KUKA KRL program: f1_Kuka_APT219T02S19.SRC

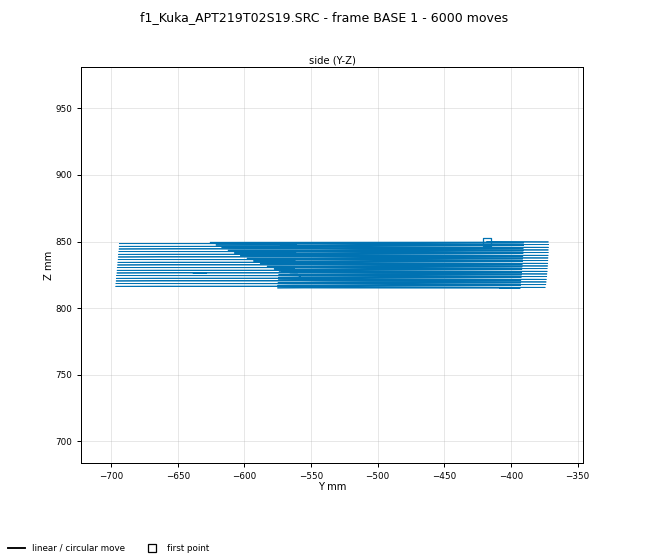
[picture p0: tool path of f1_Kuka_APT219T02S19.SRC in frame BASE 1, 6000 of 6001 moves have a stored position in this frame; points joined in program order, loops and branches not executed]
&ACCESS RVP
&REL 2
&PARAM TEMPLATE = C:\KRC\Roboter\Template\vorgabe
&PARAM EDITMASK = *
DEF f1_Kuka_APT219T02S19()


;FOLD INI;%{PE}%V3.2.0,%MKUKATPBASIS,%CINIT,%VCOMMON,%P
  ;FOLD BAS INI;%{E}%V3.2.0,%MKUKATPBASIS,%CINIT,%VINIT,%P
    GLOBAL INTERRUPT DECL 3 WHEN $STOPMESS==TRUE DO IR_STOPM ( )
    INTERRUPT ON 3
    BAS (#INITMOV,0 )
  ;ENDFOLD (BAS INI)
  ;FOLD USER INI;%{E}%V3.2.0,%MKUKATPUSER,%CINIT,%VINIT,%P
    ;Make your modifications here
  ;ENDFOLD (USER INI)
;ENDFOLD (INI)


;*** Make Null PTP Move
  PTP $pos_act

;*** Auto Load The Correct TOOL Data
  $tool=tool_data[2]

;*** Auto Load The Correct BASE Data
  $base=base_data[1]

  $ADVANCE = 5

;*** Restate Last Velocity
MMPM(30000.0)
SetRPM(8000)
LIN {X -0.097,Y -418.240,Z 849.890,A 0.000,B 0.000,C 90.000,E1 196.134} C_DIS
LIN {X -0.095,Y -415.487,Z 849.882,A 0.000,B 0.000,C 90.000,E1 194.773} C_DIS
LIN {X 0.056,Y -410.579,Z 849.869,A 0.000,B 0.000,C 90.000,E1 192.355} C_DIS
LIN {X -0.158,Y -407.973,Z 849.861,A 0.000,B 0.000,C 90.000,E1 191.007} C_DIS
LIN {X -0.079,Y -404.648,Z 849.851,A 0.000,B 0.000,C 90.000,E1 189.265} C_DIS
LIN {X -0.066,Y -401.875,Z 849.844,A 0.000,B 0.000,C 90.000,E1 187.871} C_DIS
LIN {X -0.071,Y -394.854,Z 849.822,A 0.000,B 0.000,C 90.000,E1 184.012} C_DIS
LIN {X 0.068,Y -390.052,Z 849.805,A 0.000,B 0.000,C 90.000,E1 180.802} C_DIS
LIN {X -0.073,Y -387.200,Z 849.793,A 0.000,B 0.000,C 90.000,E1 178.682} C_DIS
LIN {X 0.013,Y -383.709,Z 849.779,A 0.000,B 0.000,C 90.000,E1 176.159} C_DIS
LIN {X 0.052,Y -380.406,Z 849.765,A 0.000,B 0.000,C 90.000,E1 173.628} C_DIS
LIN {X -0.090,Y -378.246,Z 849.755,A 0.000,B 0.000,C 90.000,E1 171.837} C_DIS
LIN {X -0.103,Y -375.157,Z 849.738,A 0.000,B 0.000,C 90.000,E1 168.926} C_DIS
LIN {X -0.058,Y -372.815,Z 849.722,A 0.000,B 0.000,C 90.000,E1 165.992} C_DIS
LIN {X 0.084,Y -371.867,Z 849.706,A 0.000,B 0.000,C 90.000,E1 163.032} C_DIS
LIN {X 0.049,Y -371.826,Z 849.704,A 0.000,B 0.000,C 90.000,E1 162.670} C_DIS
LIN {X -0.054,Y -372.398,Z 849.698,A 0.000,B 0.000,C 90.000,E1 161.583} C_DIS
LIN {X -0.120,Y -372.933,Z 849.694,A 0.000,B 0.000,C 90.000,E1 160.859} C_DIS
LIN {X -0.003,Y -373.909,Z 849.690,A 0.000,B 0.000,C 90.000,E1 160.115} C_DIS
LIN {X -0.017,Y -374.079,Z 849.689,A 0.000,B 0.000,C 90.000,E1 159.934} C_DIS
LIN {X -0.070,Y -375.433,Z 849.685,A 0.000,B 0.000,C 90.000,E1 159.209} C_DIS
LIN {X 0.178,Y -376.512,Z 849.682,A 0.000,B 0.000,C 90.000,E1 158.773} C_DIS
LIN {X 0.157,Y -377.673,Z 849.680,A 0.000,B 0.000,C 90.000,E1 158.411} C_DIS
LIN {X -0.114,Y -379.654,Z 849.677,A 0.000,B 0.000,C 90.000,E1 157.922} C_DIS
LIN {X 0.023,Y -380.338,Z 849.676,A 0.000,B 0.000,C 90.000,E1 157.720} C_DIS
LIN {X -0.133,Y -381.711,Z 849.675,A 0.000,B 0.000,C 90.000,E1 157.486} C_DIS
LIN {X -0.008,Y -383.667,Z 849.673,A 0.000,B 0.000,C 90.000,E1 157.177} C_DIS
LIN {X -0.104,Y -387.727,Z 849.671,A 0.000,B 0.000,C 90.000,E1 156.719} C_DIS
LIN {X -0.011,Y -389.404,Z 849.670,A 0.000,B 0.000,C 90.000,E1 156.538} C_DIS
LIN {X -0.049,Y -392.267,Z 849.669,A 0.000,B 0.000,C 90.000,E1 156.357} C_DIS
LIN {X -0.038,Y -402.998,Z 849.666,A 0.000,B 0.000,C 90.000,E1 155.845} C_DIS
LIN {X 0.052,Y -407.988,Z 849.665,A 0.000,B 0.000,C 90.000,E1 155.665} C_DIS
LIN {X 0.056,Y -414.236,Z 849.663,A 0.000,B 0.000,C 90.000,E1 155.409} C_DIS
LIN {X -0.004,Y -424.366,Z 849.661,A 0.000,B 0.000,C 90.000,E1 154.973} C_DIS
LIN {X 0.156,Y -433.945,Z 849.658,A 0.000,B 0.000,C 90.000,E1 154.409} C_DIS
LIN {X -0.258,Y -437.088,Z 849.657,A 0.000,B 0.000,C 90.000,E1 154.280} C_DIS
LIN {X 0.137,Y -446.282,Z 849.653,A 0.000,B 0.000,C 90.000,E1 153.589} C_DIS
LIN {X -0.005,Y -452.577,Z 849.651,A 0.000,B 0.000,C 90.000,E1 153.127} C_DIS
LIN {X 0.063,Y -459.883,Z 849.647,A 0.000,B 0.000,C 90.000,E1 152.487} C_DIS
LIN {X -0.035,Y -464.270,Z 849.645,A 0.000,B 0.000,C 90.000,E1 152.103} C_DIS
LIN {X 0.201,Y -469.827,Z 849.642,A 0.000,B 0.000,C 90.000,E1 151.513} C_DIS
LIN {X -0.082,Y -478.109,Z 849.637,A 0.000,B 0.000,C 90.000,E1 150.667} C_DIS
LIN {X -0.039,Y -487.181,Z 849.631,A 0.000,B 0.000,C 90.000,E1 149.616} C_DIS
LIN {X 0.040,Y -492.120,Z 849.628,A 0.000,B 0.000,C 90.000,E1 148.997} C_DIS
LIN {X 0.149,Y -496.057,Z 849.625,A 0.000,B 0.000,C 90.000,E1 148.535} C_DIS
LIN {X 0.016,Y -498.340,Z 849.624,A 0.000,B 0.000,C 90.000,E1 148.250} C_DIS
LIN {X -0.146,Y -504.949,Z 849.619,A 0.000,B 0.000,C 90.000,E1 147.375} C_DIS
LIN {X 0.197,Y -512.229,Z 849.613,A 0.000,B 0.000,C 90.000,E1 146.294} C_DIS
LIN {X 0.024,Y -519.483,Z 849.606,A 0.000,B 0.000,C 90.000,E1 145.135} C_DIS
LIN {X -0.215,Y -527.715,Z 849.598,A 0.000,B 0.000,C 90.000,E1 143.703} C_DIS
LIN {X -0.267,Y -530.903,Z 849.595,A 0.000,B 0.000,C 90.000,E1 143.130} C_DIS
LIN {X 0.049,Y -540.478,Z 849.586,A 0.000,B 0.000,C 90.000,E1 141.376} C_DIS
LIN {X -0.271,Y -546.981,Z 849.579,A 0.000,B 0.000,C 90.000,E1 140.275} C_DIS
LIN {X 0.214,Y -551.520,Z 849.575,A 0.000,B 0.000,C 90.000,E1 139.380} C_DIS
LIN {X 0.133,Y -560.440,Z 849.565,A 0.000,B 0.000,C 90.000,E1 137.715} C_DIS
LIN {X 0.270,Y -566.970,Z 849.558,A 0.000,B 0.000,C 90.000,E1 136.458} C_DIS
LIN {X -0.153,Y -572.461,Z 849.552,A 0.000,B 0.000,C 90.000,E1 135.405} C_DIS
LIN {X 0.027,Y -580.990,Z 849.542,A 0.000,B 0.000,C 90.000,E1 133.623} C_DIS
LIN {X 0.101,Y -586.678,Z 849.536,A 0.000,B 0.000,C 90.000,E1 132.405} C_DIS
LIN {X -0.072,Y -591.498,Z 849.530,A 0.000,B 0.000,C 90.000,E1 131.353} C_DIS
LIN {X 0.072,Y -597.141,Z 849.522,A 0.000,B 0.000,C 90.000,E1 130.011} C_DIS
LIN {X 0.076,Y -601.556,Z 849.516,A 0.000,B 0.000,C 90.000,E1 128.955} C_DIS
LIN {X 0.233,Y -605.326,Z 849.511,A 0.000,B 0.000,C 90.000,E1 127.890} C_DIS
LIN {X -0.032,Y -608.724,Z 849.505,A 0.000,B 0.000,C 90.000,E1 126.870} C_DIS
LIN {X -0.043,Y -613.420,Z 849.496,A 0.000,B 0.000,C 90.000,E1 125.311} C_DIS
LIN {X -0.313,Y -614.778,Z 849.493,A 0.000,B 0.000,C 90.000,E1 124.818} C_DIS
LIN {X -0.318,Y -617.115,Z 849.488,A 0.000,B 0.000,C 90.000,E1 123.785} C_DIS
LIN {X -0.049,Y -618.145,Z 849.485,A 0.000,B 0.000,C 90.000,E1 123.245} C_DIS
LIN {X -0.026,Y -620.425,Z 849.478,A 0.000,B 0.000,C 90.000,E1 121.957} C_DIS
LIN {X 0.039,Y -622.080,Z 849.472,A 0.000,B 0.000,C 90.000,E1 120.924} C_DIS
LIN {X -0.203,Y -623.513,Z 849.466,A 0.000,B 0.000,C 90.000,E1 119.922} C_DIS
LIN {X -0.197,Y -624.516,Z 849.462,A 0.000,B 0.000,C 90.000,E1 119.155} C_DIS
LIN {X 0.148,Y -625.498,Z 849.455,A 0.000,B 0.000,C 90.000,E1 117.847} C_DIS
LIN {X 0.188,Y -625.758,Z 849.451,A 0.000,B 0.000,C 90.000,E1 117.078} C_DIS
LIN {X -0.302,Y -625.716,Z 849.443,A 0.000,B 0.000,C 90.000,E1 115.848} C_DIS
LIN {X -0.276,Y -625.442,Z 849.441,A 0.000,B 0.000,C 90.000,E1 115.335} C_DIS
LIN {X 0.313,Y -624.881,Z 849.438,A 0.000,B 0.000,C 90.000,E1 114.771} C_DIS
LIN {X 0.082,Y -623.584,Z 849.434,A 0.000,B 0.000,C 90.000,E1 114.027} C_DIS
LIN {X 0.091,Y -622.709,Z 849.431,A 0.000,B 0.000,C 90.000,E1 113.515} C_DIS
LIN {X -0.157,Y -620.296,Z 849.427,A 0.000,B 0.000,C 90.000,E1 112.898} C_DIS
LIN {X -0.180,Y -617.280,Z 849.424,A 0.000,B 0.000,C 90.000,E1 112.386} C_DIS
LIN {X -0.189,Y -616.020,Z 849.424,A 0.000,B 0.000,C 90.000,E1 112.259} C_DIS
LIN {X 0.159,Y -614.443,Z 849.423,A 0.000,B 0.000,C 90.000,E1 112.099} C_DIS
LIN {X -0.092,Y -612.293,Z 849.421,A 0.000,B 0.000,C 90.000,E1 111.844} C_DIS
LIN {X 0.060,Y -607.554,Z 849.419,A 0.000,B 0.000,C 90.000,E1 111.461} C_DIS
LIN {X 0.027,Y -606.382,Z 849.419,A 0.000,B 0.000,C 90.000,E1 111.354} C_DIS
LIN {X 0.055,Y -599.211,Z 849.416,A 0.000,B 0.000,C 90.000,E1 110.865} C_DIS
LIN {X 0.104,Y -592.657,Z 849.414,A 0.000,B 0.000,C 90.000,E1 110.482} C_DIS
LIN {X 0.085,Y -584.097,Z 849.412,A 0.000,B 0.000,C 90.000,E1 110.066} C_DIS
LIN {X 0.165,Y -569.929,Z 849.409,A 0.000,B 0.000,C 90.000,E1 109.523} C_DIS
LIN {X 0.234,Y -568.470,Z 849.408,A 0.000,B 0.000,C 90.000,E1 109.450} C_DIS
LIN {X 0.113,Y -567.497,Z 849.408,A 0.000,B 0.000,C 90.000,E1 109.396} C_DIS
LIN {X -0.170,Y -564.037,Z 849.406,A 0.000,B 0.000,C 90.000,E1 109.087} C_DIS
LIN {X -0.184,Y -563.197,Z 849.405,A 0.000,B 0.000,C 90.000,E1 108.960} C_DIS
LIN {X 0.333,Y -562.749,Z 849.405,A 0.000,B 0.000,C 90.000,E1 108.779} C_DIS
LIN {X -0.228,Y -561.358,Z 849.401,A 0.000,B 0.000,C 90.000,E1 108.236} C_DIS
LIN {X -0.207,Y -560.852,Z 849.399,A 0.000,B 0.000,C 90.000,E1 107.819} C_DIS
LIN {X 0.034,Y -560.504,Z 849.390,A 0.000,B 0.000,C 90.000,E1 106.134} C_DIS
LIN {X -0.244,Y -561.497,Z 849.373,A 0.000,B 0.000,C 90.000,E1 103.119} C_DIS
LIN {X -0.258,Y -562.639,Z 849.362,A 0.000,B 0.000,C 90.000,E1 101.186} C_DIS
LIN {X 0.207,Y -563.995,Z 849.351,A 0.000,B 0.000,C 90.000,E1 99.208} C_DIS
LIN {X -0.104,Y -565.178,Z 849.342,A 0.000,B 0.000,C 90.000,E1 97.587} C_DIS
LIN {X 0.004,Y -565.937,Z 849.334,A 0.000,B 0.000,C 90.000,E1 96.201} C_DIS
LIN {X -0.143,Y -566.362,Z 849.330,A 0.000,B 0.000,C 90.000,E1 95.391} C_DIS
LIN {X -0.083,Y -566.992,Z 849.322,A 0.000,B 0.000,C 90.000,E1 94.012} C_DIS
LIN {X 0.073,Y -567.577,Z 849.313,A 0.000,B 0.000,C 90.000,E1 92.350} C_DIS
LIN {X -0.200,Y -568.094,Z 849.302,A 0.000,B 0.000,C 90.000,E1 90.458} C_DIS
LIN {X -0.028,Y -568.457,Z 849.293,A 0.000,B 0.000,C 90.000,E1 88.797} C_DIS
LIN {X 0.038,Y -568.774,Z 849.286,A 0.000,B 0.000,C 90.000,E1 87.421} C_DIS
LIN {X 0.266,Y -569.024,Z 849.277,A 0.000,B 0.000,C 90.000,E1 85.755} C_DIS
LIN {X -0.071,Y -569.327,Z 849.268,A 0.000,B 0.000,C 90.000,E1 84.147} C_DIS
LIN {X -0.177,Y -569.742,Z 849.257,A 0.000,B 0.000,C 90.000,E1 82.243} C_DIS
LIN {X 0.182,Y -570.194,Z 849.248,A 0.000,B 0.000,C 90.000,E1 80.566} C_DIS
LIN {X -0.006,Y -570.661,Z 849.240,A 0.000,B 0.000,C 90.000,E1 79.218} C_DIS
LIN {X -0.099,Y -571.309,Z 849.231,A 0.000,B 0.000,C 90.000,E1 77.589} C_DIS
LIN {X 0.250,Y -571.898,Z 849.220,A 0.000,B 0.000,C 90.000,E1 75.644} C_DIS
LIN {X 0.022,Y -572.167,Z 849.211,A 0.000,B 0.000,C 90.000,E1 74.031} C_DIS
LIN {X -0.176,Y -572.373,Z 849.205,A 0.000,B 0.000,C 90.000,E1 72.960} C_DIS
LIN {X -0.218,Y -572.469,Z 849.196,A 0.000,B 0.000,C 90.000,E1 71.329} C_DIS
LIN {X -0.262,Y -572.329,Z 849.187,A 0.000,B 0.000,C 90.000,E1 69.699} C_DIS
LIN {X 0.061,Y -572.209,Z 849.175,A 0.000,B 0.000,C 90.000,E1 67.486} C_DIS
LIN {X 0.273,Y -572.046,Z 849.167,A 0.000,B 0.000,C 90.000,E1 66.102} C_DIS
LIN {X -0.273,Y -571.666,Z 849.160,A 0.000,B 0.000,C 90.000,E1 64.793} C_DIS
LIN {X 0.007,Y -571.054,Z 849.151,A 0.000,B 0.000,C 90.000,E1 63.127} C_DIS
LIN {X -0.060,Y -570.586,Z 849.143,A 0.000,B 0.000,C 90.000,E1 61.769} C_DIS
LIN {X 0.031,Y -570.033,Z 849.137,A 0.000,B 0.000,C 90.000,E1 60.667} C_DIS
LIN {X -0.100,Y -569.256,Z 849.131,A 0.000,B 0.000,C 90.000,E1 59.587} C_DIS
LIN {X 0.142,Y -568.528,Z 849.126,A 0.000,B 0.000,C 90.000,E1 58.742} C_DIS
LIN {X 0.108,Y -567.169,Z 849.119,A 0.000,B 0.000,C 90.000,E1 57.375} C_DIS
LIN {X -0.059,Y -565.759,Z 849.113,A 0.000,B 0.000,C 90.000,E1 56.294} C_DIS
LIN {X -0.044,Y -564.606,Z 849.108,A 0.000,B 0.000,C 90.000,E1 55.468} C_DIS
LIN {X -0.045,Y -563.349,Z 849.104,A 0.000,B 0.000,C 90.000,E1 54.642} C_DIS
LIN {X -0.085,Y -561.377,Z 849.097,A 0.000,B 0.000,C 90.000,E1 53.543} C_DIS
LIN {X -0.127,Y -559.725,Z 849.093,A 0.000,B 0.000,C 90.000,E1 52.718} C_DIS
LIN {X -0.295,Y -557.867,Z 849.088,A 0.000,B 0.000,C 90.000,E1 51.904} C_DIS
LIN {X -0.125,Y -556.538,Z 849.085,A 0.000,B 0.000,C 90.000,E1 51.331} C_DIS
LIN {X 0.029,Y -554.272,Z 849.081,A 0.000,B 0.000,C 90.000,E1 50.481} C_DIS
LIN {X 0.233,Y -551.683,Z 849.076,A 0.000,B 0.000,C 90.000,E1 49.622} C_DIS
LIN {X 0.340,Y -548.713,Z 849.071,A 0.000,B 0.000,C 90.000,E1 48.771} C_DIS
LIN {X 0.053,Y -545.404,Z 849.067,A 0.000,B 0.000,C 90.000,E1 47.957} C_DIS
LIN {X -0.123,Y -543.693,Z 849.064,A 0.000,B 0.000,C 90.000,E1 47.553} C_DIS
LIN {X 0.078,Y -540.494,Z 849.060,A 0.000,B 0.000,C 90.000,E1 46.824} C_DIS
LIN {X -0.122,Y -536.942,Z 849.056,A 0.000,B 0.000,C 90.000,E1 46.134} C_DIS
LIN {X -0.336,Y -534.702,Z 849.054,A 0.000,B 0.000,C 90.000,E1 45.729} C_DIS
LIN {X -0.216,Y -530.455,Z 849.050,A 0.000,B 0.000,C 90.000,E1 45.000} C_DIS
LIN {X -0.297,Y -526.777,Z 849.047,A 0.000,B 0.000,C 90.000,E1 44.433} C_DIS
LIN {X 0.335,Y -522.841,Z 849.044,A 0.000,B 0.000,C 90.000,E1 43.785} C_DIS
LIN {X -0.110,Y -518.541,Z 849.040,A 0.000,B 0.000,C 90.000,E1 43.257} C_DIS
LIN {X 0.016,Y -515.265,Z 849.038,A 0.000,B 0.000,C 90.000,E1 42.813} C_DIS
LIN {X -0.009,Y -510.547,Z 849.035,A 0.000,B 0.000,C 90.000,E1 42.243} C_DIS
LIN {X 0.080,Y -502.779,Z 849.030,A 0.000,B 0.000,C 90.000,E1 41.353} C_DIS
LIN {X 0.013,Y -496.096,Z 849.026,A 0.000,B 0.000,C 90.000,E1 40.663} C_DIS
LIN {X -0.057,Y -491.879,Z 849.024,A 0.000,B 0.000,C 90.000,E1 40.253} C_DIS
LIN {X -0.014,Y -486.193,Z 849.021,A 0.000,B 0.000,C 90.000,E1 39.725} C_DIS
LIN {X 0.024,Y -478.694,Z 849.017,A 0.000,B 0.000,C 90.000,E1 39.072} C_DIS
LIN {X -0.160,Y -471.068,Z 849.014,A 0.000,B 0.000,C 90.000,E1 38.463} C_DIS
LIN {X 0.188,Y -458.541,Z 849.008,A 0.000,B 0.000,C 90.000,E1 37.443} C_DIS
LIN {X -0.021,Y -450.644,Z 849.005,A 0.000,B 0.000,C 90.000,E1 36.870} C_DIS
LIN {X -0.141,Y -436.518,Z 848.999,A 0.000,B 0.000,C 90.000,E1 35.804} C_DIS
LIN {X 0.265,Y -416.517,Z 848.990,A 0.000,B 0.000,C 90.000,E1 34.119} C_DIS
LIN {X -0.154,Y -404.482,Z 848.984,A 0.000,B 0.000,C 90.000,E1 33.086} C_DIS
LIN {X 0.096,Y -399.394,Z 848.981,A 0.000,B 0.000,C 90.000,E1 32.498} C_DIS
LIN {X 0.027,Y -395.711,Z 848.978,A 0.000,B 0.000,C 90.000,E1 32.054} C_DIS
LIN {X 0.023,Y -393.423,Z 848.976,A 0.000,B 0.000,C 90.000,E1 31.592} C_DIS
LIN {X -0.137,Y -393.288,Z 848.975,A 0.000,B 0.000,C 90.000,E1 31.592} C_DIS
LIN {X -0.163,Y -393.278,Z 848.975,A 0.000,B 0.000,C 90.000,E1 31.592} C_DIS
LIN {X 0.224,Y -390.603,Z 848.968,A 0.000,B 0.000,C 90.000,E1 30.129} C_DIS
LIN {X -0.115,Y -390.372,Z 848.967,A 0.000,B 0.000,C 90.000,E1 30.001} C_DIS
LIN {X 0.019,Y -390.385,Z 848.962,A 0.000,B 0.000,C 90.000,E1 29.077} C_DIS
LIN {X -0.190,Y -391.684,Z 848.948,A 0.000,B 0.000,C 90.000,E1 26.616} C_DIS
LIN {X -0.034,Y -393.223,Z 848.936,A 0.000,B 0.000,C 90.000,E1 24.463} C_DIS
LIN {X 0.053,Y -395.280,Z 848.922,A 0.000,B 0.000,C 90.000,E1 21.972} C_DIS
LIN {X -0.118,Y -398.678,Z 848.903,A 0.000,B 0.000,C 90.000,E1 18.471} C_DIS
LIN {X -0.005,Y -402.357,Z 848.885,A 0.000,B 0.000,C 90.000,E1 15.300} C_DIS
LIN {X 0.145,Y -404.239,Z 848.877,A 0.000,B 0.000,C 90.000,E1 13.883} C_DIS
LIN {X -0.057,Y -407.324,Z 848.866,A 0.000,B 0.000,C 90.000,E1 11.827} C_DIS
LIN {X 0.131,Y -410.644,Z 848.854,A 0.000,B 0.000,C 90.000,E1 9.726} C_DIS
LIN {X -0.061,Y -415.322,Z 848.839,A 0.000,B 0.000,C 90.000,E1 7.004} C_DIS
LIN {X 0.152,Y -419.628,Z 848.826,A 0.000,B 0.000,C 90.000,E1 4.588} C_DIS
LIN {X 0.125,Y -425.733,Z 848.809,A 0.000,B 0.000,C 90.000,E1 1.547} C_DIS
LIN {X -0.196,Y -430.428,Z 848.797,A 0.000,B 0.000,C 90.000,E1 359.484} C_DIS
LIN {X -0.045,Y -436.050,Z 848.784,A 0.000,B 0.000,C 90.000,E1 357.135} C_DIS
LIN {X 0.063,Y -440.129,Z 848.775,A 0.000,B 0.000,C 90.000,E1 355.469} C_DIS
LIN {X -0.032,Y -445.378,Z 848.764,A 0.000,B 0.000,C 90.000,E1 353.514} C_DIS
LIN {X -0.133,Y -447.594,Z 848.760,A 0.000,B 0.000,C 90.000,E1 352.875} C_DIS
LIN {X 0.112,Y -449.970,Z 848.758,A 0.000,B 0.000,C 90.000,E1 352.356} C_DIS
LIN {X 0.027,Y -452.364,Z 848.756,A 0.000,B 0.000,C 90.000,E1 352.008} C_DIS
LIN {X 0.037,Y -453.322,Z 848.755,A 0.000,B 0.000,C 90.000,E1 351.894} C_DIS
LIN {X -0.122,Y -457.843,Z 848.753,A 0.000,B 0.000,C 90.000,E1 351.546} C_DIS
LIN {X 0.058,Y -464.387,Z 848.751,A 0.000,B 0.000,C 90.000,E1 351.141} C_DIS
LIN {X -0.160,Y -478.242,Z 848.747,A 0.000,B 0.000,C 90.000,E1 350.443} C_DIS
LIN {X -0.230,Y -481.631,Z 848.746,A 0.000,B 0.000,C 90.000,E1 350.274} C_DIS
LIN {X -0.042,Y -491.242,Z 848.743,A 0.000,B 0.000,C 90.000,E1 349.690} C_DIS
LIN {X 0.055,Y -503.987,Z 848.738,A 0.000,B 0.000,C 90.000,E1 348.870} C_DIS
LIN {X 0.000,Y -510.227,Z 848.736,A 0.000,B 0.000,C 90.000,E1 348.465} C_DIS
LIN {X -0.007,Y -519.606,Z 848.732,A 0.000,B 0.000,C 90.000,E1 347.825} C_DIS
LIN {X -0.120,Y -528.778,Z 848.729,A 0.000,B 0.000,C 90.000,E1 347.173} C_DIS
LIN {X -0.020,Y -539.053,Z 848.724,A 0.000,B 0.000,C 90.000,E1 346.353} C_DIS
LIN {X -0.003,Y -544.832,Z 848.722,A 0.000,B 0.000,C 90.000,E1 345.880} C_DIS
LIN {X -0.321,Y -553.121,Z 848.717,A 0.000,B 0.000,C 90.000,E1 345.172} C_DIS
LIN {X -0.213,Y -559.833,Z 848.714,A 0.000,B 0.000,C 90.000,E1 344.519} C_DIS
LIN {X -0.030,Y -564.911,Z 848.711,A 0.000,B 0.000,C 90.000,E1 343.976} C_DIS
LIN {X -0.020,Y -569.822,Z 848.708,A 0.000,B 0.000,C 90.000,E1 343.433} C_DIS
LIN {X 0.231,Y -575.816,Z 848.704,A 0.000,B 0.000,C 90.000,E1 342.725} C_DIS
LIN {X -0.110,Y -582.267,Z 848.700,A 0.000,B 0.000,C 90.000,E1 341.945} C_DIS
LIN {X -0.204,Y -588.308,Z 848.695,A 0.000,B 0.000,C 90.000,E1 341.148} C_DIS
LIN {X -0.169,Y -592.866,Z 848.692,A 0.000,B 0.000,C 90.000,E1 340.477} C_DIS
LIN {X 0.211,Y -597.895,Z 848.687,A 0.000,B 0.000,C 90.000,E1 339.645} C_DIS
LIN {X -0.276,Y -602.727,Z 848.683,A 0.000,B 0.000,C 90.000,E1 338.901} C_DIS
LIN {X -0.213,Y -608.763,Z 848.677,A 0.000,B 0.000,C 90.000,E1 337.847} C_DIS
LIN {X -0.064,Y -614.469,Z 848.671,A 0.000,B 0.000,C 90.000,E1 336.794} C_DIS
LIN {X 0.176,Y -618.529,Z 848.667,A 0.000,B 0.000,C 90.000,E1 335.997} C_DIS
LIN {X 0.142,Y -623.671,Z 848.661,A 0.000,B 0.000,C 90.000,E1 334.973} C_DIS
LIN {X -0.089,Y -628.484,Z 848.655,A 0.000,B 0.000,C 90.000,E1 333.973} C_DIS
LIN {X -0.024,Y -631.846,Z 848.651,A 0.000,B 0.000,C 90.000,E1 333.204} C_DIS
LIN {X -0.106,Y -637.026,Z 848.644,A 0.000,B 0.000,C 90.000,E1 331.948} C_DIS
LIN {X 0.106,Y -640.980,Z 848.639,A 0.000,B 0.000,C 90.000,E1 330.923} C_DIS
LIN {X 0.189,Y -645.721,Z 848.632,A 0.000,B 0.000,C 90.000,E1 329.665} C_DIS
LIN {X -0.122,Y -650.807,Z 848.623,A 0.000,B 0.000,C 90.000,E1 328.201} C_DIS
LIN {X -0.090,Y -654.566,Z 848.616,A 0.000,B 0.000,C 90.000,E1 326.962} C_DIS
LIN {X 0.000,Y -656.701,Z 848.612,A 0.000,B 0.000,C 90.000,E1 326.215} C_DIS
LIN {X 0.034,Y -659.381,Z 848.607,A 0.000,B 0.000,C 90.000,E1 325.229} C_DIS
LIN {X 0.165,Y -661.140,Z 848.603,A 0.000,B 0.000,C 90.000,E1 324.482} C_DIS
LIN {X 0.255,Y -663.369,Z 848.597,A 0.000,B 0.000,C 90.000,E1 323.497} C_DIS
LIN {X 0.338,Y -665.841,Z 848.591,A 0.000,B 0.000,C 90.000,E1 322.271} C_DIS
LIN {X -0.074,Y -668.207,Z 848.583,A 0.000,B 0.000,C 90.000,E1 320.848} C_DIS
LIN {X 0.004,Y -668.958,Z 848.580,A 0.000,B 0.000,C 90.000,E1 320.356} C_DIS
LIN {X 0.085,Y -670.549,Z 848.573,A 0.000,B 0.000,C 90.000,E1 319.138} C_DIS
LIN {X -0.170,Y -673.763,Z 848.560,A 0.000,B 0.000,C 90.000,E1 316.743} C_DIS
LIN {X 0.390,Y -674.677,Z 848.556,A 0.000,B 0.000,C 90.000,E1 315.972} C_DIS
LIN {X -0.003,Y -675.515,Z 848.552,A 0.000,B 0.000,C 90.000,E1 315.283} C_DIS
LIN {X -0.231,Y -677.518,Z 848.541,A 0.000,B 0.000,C 90.000,E1 313.380} C_DIS
LIN {X 0.055,Y -679.241,Z 848.532,A 0.000,B 0.000,C 90.000,E1 311.676} C_DIS
LIN {X 0.264,Y -680.159,Z 848.526,A 0.000,B 0.000,C 90.000,E1 310.701} C_DIS
LIN {X 0.158,Y -681.665,Z 848.517,A 0.000,B 0.000,C 90.000,E1 309.036} C_DIS
LIN {X -0.002,Y -682.710,Z 848.510,A 0.000,B 0.000,C 90.000,E1 307.855} C_DIS
LIN {X 0.006,Y -683.905,Z 848.502,A 0.000,B 0.000,C 90.000,E1 306.423} C_DIS
LIN {X 0.015,Y -684.836,Z 848.496,A 0.000,B 0.000,C 90.000,E1 305.231} C_DIS
LIN {X 0.232,Y -685.808,Z 848.488,A 0.000,B 0.000,C 90.000,E1 303.785} C_DIS
LIN {X 0.098,Y -686.998,Z 848.479,A 0.000,B 0.000,C 90.000,E1 302.133} C_DIS
LIN {X 0.054,Y -688.571,Z 848.467,A 0.000,B 0.000,C 90.000,E1 300.001} C_DIS
LIN {X -0.146,Y -689.928,Z 848.458,A 0.000,B 0.000,C 90.000,E1 298.359} C_DIS
LIN {X 0.044,Y -691.166,Z 848.450,A 0.000,B 0.000,C 90.000,E1 296.924} C_DIS
LIN {X 0.319,Y -692.286,Z 848.443,A 0.000,B 0.000,C 90.000,E1 295.720} C_DIS
LIN {X 0.372,Y -693.183,Z 848.438,A 0.000,B 0.000,C 90.000,E1 294.771} C_DIS
LIN {X 0.189,Y -693.660,Z 848.434,A 0.000,B 0.000,C 90.000,E1 294.079} C_DIS
LIN {X 0.434,Y -693.784,Z 848.433,A 0.000,B 0.000,C 90.000,E1 293.823} C_DIS
LIN {X 0.010,Y -693.649,Z 848.430,A 0.000,B 0.000,C 90.000,E1 293.387} C_DIS
LIN {X -0.020,Y -693.448,Z 848.429,A 0.000,B 0.000,C 90.000,E1 293.153} C_DIS
LIN {X -0.173,Y -691.784,Z 848.426,A 0.000,B 0.000,C 90.000,E1 292.695} C_DIS
LIN {X -0.202,Y -690.736,Z 848.425,A 0.000,B 0.000,C 90.000,E1 292.461} C_DIS
LIN {X -0.085,Y -689.821,Z 848.424,A 0.000,B 0.000,C 90.000,E1 292.333} C_DIS
LIN {X 0.259,Y -684.750,Z 848.422,A 0.000,B 0.000,C 90.000,E1 291.844} C_DIS
LIN {X -0.187,Y -683.162,Z 848.421,A 0.000,B 0.000,C 90.000,E1 291.770} C_DIS
LIN {X -0.103,Y -680.903,Z 848.420,A 0.000,B 0.000,C 90.000,E1 291.663} C_DIS
LIN {X -0.201,Y -671.049,Z 848.418,A 0.000,B 0.000,C 90.000,E1 291.334} C_DIS
LIN {X 0.301,Y -662.762,Z 848.417,A 0.000,B 0.000,C 90.000,E1 291.099} C_DIS
LIN {X 0.107,Y -655.161,Z 848.417,A 0.000,B 0.000,C 90.000,E1 290.972} C_DIS
LIN {X 0.014,Y -647.937,Z 848.416,A 0.000,B 0.000,C 90.000,E1 290.791} C_DIS
LIN {X 0.301,Y -644.900,Z 848.415,A 0.000,B 0.000,C 90.000,E1 290.663} C_DIS
LIN {X -0.053,Y -638.911,Z 848.414,A 0.000,B 0.000,C 90.000,E1 290.429} C_DIS
LIN {X -0.362,Y -636.284,Z 848.412,A 0.000,B 0.000,C 90.000,E1 290.248} C_DIS
LIN {X 0.197,Y -636.268,Z 848.412,A 0.000,B 0.000,C 90.000,E1 290.194} C_DIS
LIN {X -0.021,Y -636.024,Z 848.412,A 0.000,B 0.000,C 90.000,E1 290.120} C_DIS
LIN {X 0.171,Y -637.336,Z 848.409,A 0.000,B 0.000,C 90.000,E1 289.631} C_DIS
LIN {X -0.057,Y -641.499,Z 848.405,A 0.000,B 0.000,C 90.000,E1 288.852} C_DIS
LIN {X -0.161,Y -644.934,Z 848.401,A 0.000,B 0.000,C 90.000,E1 288.236} C_DIS
LIN {X 0.200,Y -648.505,Z 848.397,A 0.000,B 0.000,C 90.000,E1 287.457} C_DIS
LIN {X -0.082,Y -650.705,Z 848.394,A 0.000,B 0.000,C 90.000,E1 286.985} C_DIS
LIN {X -0.288,Y -653.598,Z 848.390,A 0.000,B 0.000,C 90.000,E1 286.260} C_DIS
LIN {X 0.097,Y -655.375,Z 848.388,A 0.000,B 0.000,C 90.000,E1 285.733} C_DIS
LIN {X -0.072,Y -657.543,Z 848.383,A 0.000,B 0.000,C 90.000,E1 285.009} C_DIS
LIN {X -0.290,Y -658.737,Z 848.381,A 0.000,B 0.000,C 90.000,E1 284.537} C_DIS
LIN {X 0.040,Y -660.004,Z 848.377,A 0.000,B 0.000,C 90.000,E1 283.772} C_DIS
LIN {X -0.160,Y -660.688,Z 848.374,A 0.000,B 0.000,C 90.000,E1 283.300} C_DIS
LIN {X 0.289,Y -661.199,Z 848.371,A 0.000,B 0.000,C 90.000,E1 282.771} C_DIS
LIN {X -0.001,Y -661.523,Z 848.367,A 0.000,B 0.000,C 90.000,E1 282.063} C_DIS
LIN {X -0.196,Y -661.470,Z 848.364,A 0.000,B 0.000,C 90.000,E1 281.591} C_DIS
LIN {X 0.126,Y -661.223,Z 848.362,A 0.000,B 0.000,C 90.000,E1 281.074} C_DIS
LIN {X -0.174,Y -660.488,Z 848.358,A 0.000,B 0.000,C 90.000,E1 280.366} C_DIS
LIN {X 0.153,Y -659.752,Z 848.355,A 0.000,B 0.000,C 90.000,E1 279.849} C_DIS
LIN {X -0.063,Y -658.593,Z 848.352,A 0.000,B 0.000,C 90.000,E1 279.378} C_DIS
LIN {X 0.256,Y -657.119,Z 848.349,A 0.000,B 0.000,C 90.000,E1 278.859} C_DIS
LIN {X -0.081,Y -655.281,Z 848.347,A 0.000,B 0.000,C 90.000,E1 278.398} C_DIS
LIN {X 0.313,Y -653.075,Z 848.344,A 0.000,B 0.000,C 90.000,E1 277.871} C_DIS
LIN {X -0.021,Y -651.178,Z 848.342,A 0.000,B 0.000,C 90.000,E1 277.530} C_DIS
LIN {X 0.255,Y -648.349,Z 848.339,A 0.000,B 0.000,C 90.000,E1 277.011} C_DIS
LIN {X -0.016,Y -646.062,Z 848.337,A 0.000,B 0.000,C 90.000,E1 276.663} C_DIS
LIN {X 0.099,Y -641.432,Z 848.334,A 0.000,B 0.000,C 90.000,E1 276.030} C_DIS
LIN {X -0.329,Y -637.002,Z 848.331,A 0.000,B 0.000,C 90.000,E1 275.568} C_DIS
LIN {X -0.023,Y -631.916,Z 848.328,A 0.000,B 0.000,C 90.000,E1 275.049} C_DIS
LIN {X 0.028,Y -626.134,Z 848.326,A 0.000,B 0.000,C 90.000,E1 274.588} C_DIS
LIN {X 0.174,Y -623.067,Z 848.324,A 0.000,B 0.000,C 90.000,E1 274.359} C_DIS
LIN {X 0.004,Y -618.447,Z 848.323,A 0.000,B 0.000,C 90.000,E1 274.073} C_DIS
LIN {X 0.122,Y -610.631,Z 848.320,A 0.000,B 0.000,C 90.000,E1 273.612} C_DIS
LIN {X 0.218,Y -603.841,Z 848.318,A 0.000,B 0.000,C 90.000,E1 273.269} C_DIS
LIN {X 0.022,Y -596.974,Z 848.317,A 0.000,B 0.000,C 90.000,E1 272.980} C_DIS
LIN {X 0.207,Y -591.698,Z 848.315,A 0.000,B 0.000,C 90.000,E1 272.751} C_DIS
LIN {X 0.032,Y -584.016,Z 848.314,A 0.000,B 0.000,C 90.000,E1 272.522} C_DIS
LIN {X 0.250,Y -577.825,Z 848.313,A 0.000,B 0.000,C 90.000,E1 272.350} C_DIS
LIN {X -0.171,Y -570.988,Z 848.313,A 0.000,B 0.000,C 90.000,E1 272.293} C_DIS
LIN {X -0.136,Y -564.922,Z 848.312,A 0.000,B 0.000,C 90.000,E1 272.236} C_DIS
LIN {X 0.235,Y -557.839,Z 848.312,A 0.000,B 0.000,C 90.000,E1 272.178} C_DIS
LIN {X -0.118,Y -553.030,Z 848.312,A 0.000,B 0.000,C 90.000,E1 272.178} C_DIS
LIN {X -0.048,Y -549.930,Z 848.311,A 0.000,B 0.000,C 90.000,E1 272.064} C_DIS
LIN {X -0.085,Y -549.889,Z 848.311,A 0.000,B 0.000,C 90.000,E1 272.064} C_DIS
LIN {X -0.036,Y -548.958,Z 848.311,A 0.000,B 0.000,C 90.000,E1 271.892} C_DIS
LIN {X -0.136,Y -547.957,Z 848.309,A 0.000,B 0.000,C 90.000,E1 271.604} C_DIS
LIN {X 0.022,Y -546.966,Z 848.306,A 0.000,B 0.000,C 90.000,E1 271.031} C_DIS
LIN {X 0.156,Y -546.102,Z 848.301,A 0.000,B 0.000,C 90.000,E1 270.172} C_DIS
LIN {X -0.114,Y -544.536,Z 848.290,A 0.000,B 0.000,C 90.000,E1 268.224} C_DIS
LIN {X 0.098,Y -543.579,Z 848.282,A 0.000,B 0.000,C 90.000,E1 266.788} C_DIS
LIN {X -0.213,Y -542.395,Z 848.273,A 0.000,B 0.000,C 90.000,E1 265.122} C_DIS
LIN {X 0.038,Y -541.177,Z 848.263,A 0.000,B 0.000,C 90.000,E1 263.394} C_DIS
LIN {X -0.222,Y -539.365,Z 848.252,A 0.000,B 0.000,C 90.000,E1 261.432} C_DIS
LIN {X 0.028,Y -538.065,Z 848.244,A 0.000,B 0.000,C 90.000,E1 259.982} C_DIS
LIN {X -0.115,Y -536.335,Z 848.235,A 0.000,B 0.000,C 90.000,E1 258.285} C_DIS
LIN {X 0.117,Y -535.199,Z 848.229,A 0.000,B 0.000,C 90.000,E1 257.117} C_DIS
LIN {X -0.019,Y -533.454,Z 848.221,A 0.000,B 0.000,C 90.000,E1 255.700} C_DIS
LIN {X -0.009,Y -531.474,Z 848.211,A 0.000,B 0.000,C 90.000,E1 253.976} C_DIS
LIN {X -0.095,Y -530.108,Z 848.205,A 0.000,B 0.000,C 90.000,E1 252.834} C_DIS
LIN {X -0.186,Y -528.341,Z 848.197,A 0.000,B 0.000,C 90.000,E1 251.402} C_DIS
LIN {X 0.025,Y -526.478,Z 848.189,A 0.000,B 0.000,C 90.000,E1 249.934} C_DIS
LIN {X 0.206,Y -524.511,Z 848.181,A 0.000,B 0.000,C 90.000,E1 248.465} C_DIS
LIN {X 0.015,Y -522.006,Z 848.171,A 0.000,B 0.000,C 90.000,E1 246.741} C_DIS
LIN {X -0.329,Y -520.282,Z 848.164,A 0.000,B 0.000,C 90.000,E1 245.613} C_DIS
LIN {X -0.009,Y -518.460,Z 848.158,A 0.000,B 0.000,C 90.000,E1 244.409} C_DIS
LIN {X -0.158,Y -515.412,Z 848.148,A 0.000,B 0.000,C 90.000,E1 242.666} C_DIS
LIN {X 0.077,Y -512.292,Z 848.138,A 0.000,B 0.000,C 90.000,E1 240.873} C_DIS
LIN {X -0.035,Y -510.717,Z 848.133,A 0.000,B 0.000,C 90.000,E1 239.999} C_DIS
LIN {X 0.139,Y -507.372,Z 848.123,A 0.000,B 0.000,C 90.000,E1 238.201} C_DIS
LIN {X -0.128,Y -505.065,Z 848.117,A 0.000,B 0.000,C 90.000,E1 237.041} C_DIS
LIN {X 0.270,Y -502.502,Z 848.110,A 0.000,B 0.000,C 90.000,E1 235.801} C_DIS
LIN {X 0.093,Y -499.182,Z 848.102,A 0.000,B 0.000,C 90.000,E1 234.322} C_DIS
LIN {X -0.013,Y -492.749,Z 848.087,A 0.000,B 0.000,C 90.000,E1 231.618} C_DIS
LIN {X -0.307,Y -489.893,Z 848.080,A 0.000,B 0.000,C 90.000,E1 230.436} C_DIS
LIN {X 0.042,Y -487.094,Z 848.073,A 0.000,B 0.000,C 90.000,E1 229.175} C_DIS
LIN {X 0.059,Y -482.174,Z 848.061,A 0.000,B 0.000,C 90.000,E1 227.025} C_DIS
LIN {X 0.035,Y -476.902,Z 848.048,A 0.000,B 0.000,C 90.000,E1 224.555} C_DIS
LIN {X -0.075,Y -475.530,Z 848.044,A 0.000,B 0.000,C 90.000,E1 223.947} C_DIS
LIN {X -0.122,Y -471.482,Z 848.034,A 0.000,B 0.000,C 90.000,E1 222.081} C_DIS
LIN {X 0.021,Y -468.104,Z 848.025,A 0.000,B 0.000,C 90.000,E1 220.496} C_DIS
LIN {X 0.096,Y -464.800,Z 848.016,A 0.000,B 0.000,C 90.000,E1 218.910} C_DIS
LIN {X 0.057,Y -462.199,Z 848.009,A 0.000,B 0.000,C 90.000,E1 217.649} C_DIS
LIN {X 0.184,Y -458.215,Z 847.999,A 0.000,B 0.000,C 90.000,E1 215.724} C_DIS
LIN {X 0.226,Y -454.739,Z 847.990,A 0.000,B 0.000,C 90.000,E1 214.119} C_DIS
LIN {X 0.126,Y -449.913,Z 847.977,A 0.000,B 0.000,C 90.000,E1 211.878} C_DIS
LIN {X 0.136,Y -446.480,Z 847.968,A 0.000,B 0.000,C 90.000,E1 210.256} C_DIS
LIN {X 0.079,Y -442.509,Z 847.957,A 0.000,B 0.000,C 90.000,E1 208.309} C_DIS
LIN {X -0.036,Y -437.834,Z 847.945,A 0.000,B 0.000,C 90.000,E1 206.027} C_DIS
LIN {X -0.114,Y -434.513,Z 847.935,A 0.000,B 0.000,C 90.000,E1 204.387} C_DIS
LIN {X -0.031,Y -431.126,Z 847.926,A 0.000,B 0.000,C 90.000,E1 202.717} C_DIS
LIN {X 0.003,Y -426.544,Z 847.913,A 0.000,B 0.000,C 90.000,E1 200.375} C_DIS
LIN {X 0.153,Y -422.001,Z 847.900,A 0.000,B 0.000,C 90.000,E1 198.000} C_DIS
LIN {X 0.146,Y -418.069,Z 847.889,A 0.000,B 0.000,C 90.000,E1 195.969} C_DIS
LIN {X -0.146,Y -415.336,Z 847.881,A 0.000,B 0.000,C 90.000,E1 194.647} C_DIS
LIN {X -0.094,Y -410.450,Z 847.868,A 0.000,B 0.000,C 90.000,E1 192.243} C_DIS
LIN {X 0.072,Y -408.497,Z 847.862,A 0.000,B 0.000,C 90.000,E1 191.186} C_DIS
LIN {X 0.164,Y -405.188,Z 847.853,A 0.000,B 0.000,C 90.000,E1 189.443} C_DIS
LIN {X 0.191,Y -402.483,Z 847.845,A 0.000,B 0.000,C 90.000,E1 188.049} C_DIS
LIN {X -0.105,Y -395.915,Z 847.825,A 0.000,B 0.000,C 90.000,E1 184.588} C_DIS
LIN {X -0.157,Y -392.032,Z 847.812,A 0.000,B 0.000,C 90.000,E1 182.121} C_DIS
LIN {X -0.027,Y -388.097,Z 847.796,A 0.000,B 0.000,C 90.000,E1 179.255} C_DIS
LIN {X 0.090,Y -386.661,Z 847.790,A 0.000,B 0.000,C 90.000,E1 178.165} C_DIS
LIN {X 0.169,Y -383.238,Z 847.776,A 0.000,B 0.000,C 90.000,E1 175.641} C_DIS
LIN {X -0.181,Y -380.038,Z 847.762,A 0.000,B 0.000,C 90.000,E1 173.166} C_DIS
LIN {X -0.159,Y -377.072,Z 847.748,A 0.000,B 0.000,C 90.000,E1 170.622} C_DIS
LIN {X 0.120,Y -375.244,Z 847.738,A 0.000,B 0.000,C 90.000,E1 168.757} C_DIS
LIN {X -0.082,Y -373.168,Z 847.723,A 0.000,B 0.000,C 90.000,E1 166.228} C_DIS
LIN {X 0.036,Y -371.759,Z 847.705,A 0.000,B 0.000,C 90.000,E1 162.906} C_DIS
LIN {X 0.001,Y -371.728,Z 847.703,A 0.000,B 0.000,C 90.000,E1 162.543} C_DIS
LIN {X -0.134,Y -372.416,Z 847.695,A 0.000,B 0.000,C 90.000,E1 161.094} C_DIS
LIN {X -0.230,Y -373.403,Z 847.689,A 0.000,B 0.000,C 90.000,E1 160.007} C_DIS
LIN {X -0.187,Y -375.174,Z 847.683,A 0.000,B 0.000,C 90.000,E1 158.901} C_DIS
LIN {X -0.099,Y -376.948,Z 847.679,A 0.000,B 0.000,C 90.000,E1 158.156} C_DIS
LIN {X -0.131,Y -378.660,Z 847.676,A 0.000,B 0.000,C 90.000,E1 157.614} C_DIS
LIN {X -0.059,Y -380.504,Z 847.673,A 0.000,B 0.000,C 90.000,E1 157.177} C_DIS
LIN {X 0.084,Y -381.357,Z 847.672,A 0.000,B 0.000,C 90.000,E1 156.975} C_DIS
LIN {X 0.040,Y -383.255,Z 847.670,A 0.000,B 0.000,C 90.000,E1 156.666} C_DIS
LIN {X -0.045,Y -386.426,Z 847.668,A 0.000,B 0.000,C 90.000,E1 156.305} C_DIS
LIN {X 0.040,Y -390.790,Z 847.666,A 0.000,B 0.000,C 90.000,E1 155.869} C_DIS
LIN {X -0.226,Y -399.042,Z 847.664,A 0.000,B 0.000,C 90.000,E1 155.485} C_DIS
LIN {X -0.069,Y -404.850,Z 847.662,A 0.000,B 0.000,C 90.000,E1 155.229} C_DIS
LIN {X -0.163,Y -408.741,Z 847.662,A 0.000,B 0.000,C 90.000,E1 155.101} C_DIS
LIN {X 0.043,Y -422.514,Z 847.658,A 0.000,B 0.000,C 90.000,E1 154.485} C_DIS
LIN {X 0.034,Y -432.152,Z 847.655,A 0.000,B 0.000,C 90.000,E1 153.973} C_DIS
LIN {X 0.019,Y -438.603,Z 847.653,A 0.000,B 0.000,C 90.000,E1 153.589} C_DIS
LIN {X -0.011,Y -449.485,Z 847.649,A 0.000,B 0.000,C 90.000,E1 152.820} C_DIS
LIN {X -0.133,Y -453.874,Z 847.647,A 0.000,B 0.000,C 90.000,E1 152.487} C_DIS
LIN {X -0.136,Y -459.944,Z 847.644,A 0.000,B 0.000,C 90.000,E1 151.975} C_DIS
LIN {X -0.010,Y -469.830,Z 847.639,A 0.000,B 0.000,C 90.000,E1 151.001} C_DIS
LIN {X -0.260,Y -475.228,Z 847.636,A 0.000,B 0.000,C 90.000,E1 150.461} C_DIS
LIN {X 0.134,Y -481.730,Z 847.632,A 0.000,B 0.000,C 90.000,E1 149.665} C_DIS
LIN {X 0.077,Y -484.281,Z 847.630,A 0.000,B 0.000,C 90.000,E1 149.410} C_DIS
LIN {X 0.144,Y -490.454,Z 847.626,A 0.000,B 0.000,C 90.000,E1 148.663} C_DIS
LIN {X -0.170,Y -493.048,Z 847.624,A 0.000,B 0.000,C 90.000,E1 148.408} C_DIS
LIN {X 0.182,Y -496.678,Z 847.622,A 0.000,B 0.000,C 90.000,E1 147.916} C_DIS
LIN {X -0.079,Y -503.225,Z 847.617,A 0.000,B 0.000,C 90.000,E1 147.041} C_DIS
LIN {X 0.006,Y -509.665,Z 847.612,A 0.000,B 0.000,C 90.000,E1 146.135} C_DIS
LIN {X -0.017,Y -516.050,Z 847.606,A 0.000,B 0.000,C 90.000,E1 145.102} C_DIS
LIN {X 0.116,Y -524.473,Z 847.598,A 0.000,B 0.000,C 90.000,E1 143.623} C_DIS
LIN {X 0.017,Y -529.430,Z 847.593,A 0.000,B 0.000,C 90.000,E1 142.763} C_DIS
LIN {X 0.130,Y -536.755,Z 847.586,A 0.000,B 0.000,C 90.000,E1 141.457} C_DIS
LIN {X -0.243,Y -543.294,Z 847.580,A 0.000,B 0.000,C 90.000,E1 140.356} C_DIS
LIN {X -0.177,Y -549.411,Z 847.573,A 0.000,B 0.000,C 90.000,E1 139.218} C_DIS
LIN {X -0.307,Y -558.313,Z 847.564,A 0.000,B 0.000,C 90.000,E1 137.553} C_DIS
LIN {X -0.208,Y -564.890,Z 847.557,A 0.000,B 0.000,C 90.000,E1 136.296} C_DIS
LIN {X -0.107,Y -569.687,Z 847.552,A 0.000,B 0.000,C 90.000,E1 135.324} C_DIS
LIN {X -0.055,Y -573.065,Z 847.548,A 0.000,B 0.000,C 90.000,E1 134.636} C_DIS
LIN {X 0.294,Y -576.902,Z 847.543,A 0.000,B 0.000,C 90.000,E1 133.785} C_DIS
LIN {X 0.149,Y -581.424,Z 847.538,A 0.000,B 0.000,C 90.000,E1 132.852} C_DIS
LIN {X 0.060,Y -585.803,Z 847.533,A 0.000,B 0.000,C 90.000,E1 131.919} C_DIS
LIN {X 0.014,Y -589.876,Z 847.528,A 0.000,B 0.000,C 90.000,E1 130.987} C_DIS
LIN {X 0.135,Y -595.523,Z 847.520,A 0.000,B 0.000,C 90.000,E1 129.644} C_DIS
LIN {X 0.349,Y -598.761,Z 847.516,A 0.000,B 0.000,C 90.000,E1 128.830} C_DIS
LIN {X -0.248,Y -601.703,Z 847.512,A 0.000,B 0.000,C 90.000,E1 128.096} C_DIS
LIN {X 0.026,Y -604.360,Z 847.507,A 0.000,B 0.000,C 90.000,E1 127.282} C_DIS
LIN {X 0.226,Y -607.499,Z 847.501,A 0.000,B 0.000,C 90.000,E1 126.217} C_DIS
LIN {X 0.120,Y -610.444,Z 847.496,A 0.000,B 0.000,C 90.000,E1 125.185} C_DIS
LIN {X 0.120,Y -612.289,Z 847.491,A 0.000,B 0.000,C 90.000,E1 124.405} C_DIS
LIN {X 0.131,Y -613.913,Z 847.487,A 0.000,B 0.000,C 90.000,E1 123.627} C_DIS
LIN {X -0.222,Y -615.695,Z 847.481,A 0.000,B 0.000,C 90.000,E1 122.625} C_DIS
LIN {X -0.220,Y -617.333,Z 847.475,A 0.000,B 0.000,C 90.000,E1 121.592} C_DIS
LIN {X 0.008,Y -618.752,Z 847.470,A 0.000,B 0.000,C 90.000,E1 120.541} C_DIS
LIN {X -0.274,Y -620.017,Z 847.464,A 0.000,B 0.000,C 90.000,E1 119.539} C_DIS
LIN {X -0.010,Y -621.093,Z 847.457,A 0.000,B 0.000,C 90.000,E1 118.231} C_DIS
LIN {X -0.013,Y -621.270,Z 847.455,A 0.000,B 0.000,C 90.000,E1 117.975} C_DIS
LIN {X -0.017,Y -621.368,Z 847.451,A 0.000,B 0.000,C 90.000,E1 117.206} C_DIS
LIN {X -0.017,Y -621.292,Z 847.445,A 0.000,B 0.000,C 90.000,E1 116.181} C_DIS
LIN {X -0.020,Y -620.759,Z 847.441,A 0.000,B 0.000,C 90.000,E1 115.412} C_DIS
LIN {X -0.026,Y -620.224,Z 847.438,A 0.000,B 0.000,C 90.000,E1 114.899} C_DIS
LIN {X -0.048,Y -618.867,Z 847.434,A 0.000,B 0.000,C 90.000,E1 114.131} C_DIS
LIN {X -0.323,Y -617.721,Z 847.431,A 0.000,B 0.000,C 90.000,E1 113.643} C_DIS
LIN {X 0.211,Y -616.168,Z 847.428,A 0.000,B 0.000,C 90.000,E1 113.078} C_DIS
LIN {X 0.199,Y -615.432,Z 847.428,A 0.000,B 0.000,C 90.000,E1 112.950} C_DIS
LIN {X -0.312,Y -613.941,Z 847.426,A 0.000,B 0.000,C 90.000,E1 112.642} C_DIS
LIN {X 0.240,Y -613.246,Z 847.425,A 0.000,B 0.000,C 90.000,E1 112.461} C_DIS
LIN {X -0.324,Y -609.469,Z 847.422,A 0.000,B 0.000,C 90.000,E1 112.025} C_DIS
LIN {X -0.177,Y -606.429,Z 847.421,A 0.000,B 0.000,C 90.000,E1 111.770} C_DIS
LIN {X -0.225,Y -604.092,Z 847.420,A 0.000,B 0.000,C 90.000,E1 111.535} C_DIS
LIN {X -0.052,Y -600.876,Z 847.418,A 0.000,B 0.000,C 90.000,E1 111.280} C_DIS
LIN {X -0.218,Y -596.295,Z 847.416,A 0.000,B 0.000,C 90.000,E1 110.972} C_DIS
LIN {X 0.058,Y -589.730,Z 847.414,A 0.000,B 0.000,C 90.000,E1 110.556} C_DIS
LIN {X -0.301,Y -582.578,Z 847.412,A 0.000,B 0.000,C 90.000,E1 110.248} C_DIS
LIN {X -0.001,Y -570.851,Z 847.410,A 0.000,B 0.000,C 90.000,E1 109.758} C_DIS
LIN {X 0.018,Y -569.364,Z 847.409,A 0.000,B 0.000,C 90.000,E1 109.685} C_DIS
LIN {X 0.023,Y -566.756,Z 847.408,A 0.000,B 0.000,C 90.000,E1 109.504} C_DIS
LIN {X 0.241,Y -564.570,Z 847.407,A 0.000,B 0.000,C 90.000,E1 109.268} C_DIS
LIN {X 0.173,Y -563.781,Z 847.406,A 0.000,B 0.000,C 90.000,E1 109.141} C_DIS
LIN {X -0.185,Y -562.807,Z 847.405,A 0.000,B 0.000,C 90.000,E1 108.906} C_DIS
LIN {X -0.126,Y -561.565,Z 847.402,A 0.000,B 0.000,C 90.000,E1 108.290} C_DIS
LIN {X 0.317,Y -560.985,Z 847.398,A 0.000,B 0.000,C 90.000,E1 107.692} C_DIS
LIN {X 0.002,Y -560.727,Z 847.388,A 0.000,B 0.000,C 90.000,E1 105.788} C_DIS
LIN {X 0.144,Y -561.743,Z 847.372,A 0.000,B 0.000,C 90.000,E1 103.008} C_DIS
LIN {X -0.248,Y -563.074,Z 847.360,A 0.000,B 0.000,C 90.000,E1 100.838} C_DIS
LIN {X 0.068,Y -564.228,Z 847.351,A 0.000,B 0.000,C 90.000,E1 99.151} C_DIS
LIN {X 0.237,Y -565.220,Z 847.343,A 0.000,B 0.000,C 90.000,E1 97.757} C_DIS
LIN {X 0.182,Y -565.881,Z 847.337,A 0.000,B 0.000,C 90.000,E1 96.663} C_DIS
LIN {X 0.296,Y -566.593,Z 847.330,A 0.000,B 0.000,C 90.000,E1 95.277} C_DIS
LIN {X -0.201,Y -567.223,Z 847.322,A 0.000,B 0.000,C 90.000,E1 93.955} C_DIS
LIN {X -0.039,Y -567.795,Z 847.313,A 0.000,B 0.000,C 90.000,E1 92.293} C_DIS
LIN {X 0.261,Y -568.312,Z 847.302,A 0.000,B 0.000,C 90.000,E1 90.344} C_DIS
LIN {X -0.131,Y -568.698,Z 847.293,A 0.000,B 0.000,C 90.000,E1 88.740} C_DIS
LIN {X 0.061,Y -569.055,Z 847.284,A 0.000,B 0.000,C 90.000,E1 87.078} C_DIS
LIN {X -0.277,Y -569.292,Z 847.275,A 0.000,B 0.000,C 90.000,E1 85.469} C_DIS
LIN {X -0.162,Y -569.575,Z 847.267,A 0.000,B 0.000,C 90.000,E1 84.090} C_DIS
LIN {X -0.265,Y -569.982,Z 847.256,A 0.000,B 0.000,C 90.000,E1 82.186} C_DIS
LIN {X 0.190,Y -570.425,Z 847.247,A 0.000,B 0.000,C 90.000,E1 80.500} C_DIS
LIN {X -0.089,Y -570.903,Z 847.240,A 0.000,B 0.000,C 90.000,E1 79.162} C_DIS
LIN {X -0.058,Y -571.515,Z 847.231,A 0.000,B 0.000,C 90.000,E1 77.521} C_DIS
LIN {X 0.169,Y -572.093,Z 847.220,A 0.000,B 0.000,C 90.000,E1 75.589} C_DIS
LIN {X -0.059,Y -572.360,Z 847.211,A 0.000,B 0.000,C 90.000,E1 73.976} C_DIS
LIN {X -0.258,Y -572.527,Z 847.205,A 0.000,B 0.000,C 90.000,E1 72.906} C_DIS
LIN {X 0.241,Y -572.597,Z 847.196,A 0.000,B 0.000,C 90.000,E1 71.221} C_DIS
LIN {X -0.149,Y -572.470,Z 847.187,A 0.000,B 0.000,C 90.000,E1 69.625} C_DIS
LIN {X 0.188,Y -572.292,Z 847.175,A 0.000,B 0.000,C 90.000,E1 67.411} C_DIS
LIN {X 0.177,Y -572.088,Z 847.167,A 0.000,B 0.000,C 90.000,E1 66.049} C_DIS
LIN {X -0.130,Y -571.678,Z 847.159,A 0.000,B 0.000,C 90.000,E1 64.717} C_DIS
LIN {X -0.099,Y -571.045,Z 847.150,A 0.000,B 0.000,C 90.000,E1 63.076} C_DIS
LIN {X 0.097,Y -570.557,Z 847.143,A 0.000,B 0.000,C 90.000,E1 61.691} C_DIS
LIN {X 0.191,Y -569.987,Z 847.137,A 0.000,B 0.000,C 90.000,E1 60.589} C_DIS
LIN {X -0.048,Y -569.403,Z 847.132,A 0.000,B 0.000,C 90.000,E1 59.793} C_DIS
LIN {X 0.307,Y -568.391,Z 847.126,A 0.000,B 0.000,C 90.000,E1 58.663} C_DIS
LIN {X -0.032,Y -566.983,Z 847.119,A 0.000,B 0.000,C 90.000,E1 57.327} C_DIS
LIN {X 0.108,Y -565.541,Z 847.112,A 0.000,B 0.000,C 90.000,E1 56.215} C_DIS
LIN {X 0.122,Y -564.354,Z 847.108,A 0.000,B 0.000,C 90.000,E1 55.388} C_DIS
LIN {X 0.120,Y -563.065,Z 847.103,A 0.000,B 0.000,C 90.000,E1 54.562} C_DIS
LIN {X -0.023,Y -561.593,Z 847.099,A 0.000,B 0.000,C 90.000,E1 53.749} C_DIS
LIN {X -0.060,Y -559.963,Z 847.094,A 0.000,B 0.000,C 90.000,E1 52.924} C_DIS
LIN {X -0.138,Y -557.405,Z 847.088,A 0.000,B 0.000,C 90.000,E1 51.823} C_DIS
LIN {X 0.030,Y -556.068,Z 847.085,A 0.000,B 0.000,C 90.000,E1 51.251} C_DIS
LIN {X -0.173,Y -553.712,Z 847.080,A 0.000,B 0.000,C 90.000,E1 50.436} C_DIS
LIN {X 0.316,Y -551.989,Z 847.077,A 0.000,B 0.000,C 90.000,E1 49.828} C_DIS
LIN {X 0.068,Y -549.063,Z 847.072,A 0.000,B 0.000,C 90.000,E1 49.013} C_DIS
LIN {X 0.150,Y -545.794,Z 847.068,A 0.000,B 0.000,C 90.000,E1 48.162} C_DIS
LIN {X 0.004,Y -542.839,Z 847.064,A 0.000,B 0.000,C 90.000,E1 47.472} C_DIS
LIN {X -0.173,Y -539.565,Z 847.060,A 0.000,B 0.000,C 90.000,E1 46.782} C_DIS
LIN {X -0.193,Y -536.719,Z 847.057,A 0.000,B 0.000,C 90.000,E1 46.215} C_DIS
LIN {X -0.232,Y -533.615,Z 847.054,A 0.000,B 0.000,C 90.000,E1 45.648} C_DIS
LIN {X -0.291,Y -530.187,Z 847.050,A 0.000,B 0.000,C 90.000,E1 45.081} C_DIS
LIN {X -0.212,Y -525.436,Z 847.046,A 0.000,B 0.000,C 90.000,E1 44.352} C_DIS
LIN {X 0.257,Y -522.466,Z 847.044,A 0.000,B 0.000,C 90.000,E1 43.866} C_DIS
LIN {X -0.100,Y -516.926,Z 847.040,A 0.000,B 0.000,C 90.000,E1 43.176} C_DIS
LIN {X 0.018,Y -513.528,Z 847.037,A 0.000,B 0.000,C 90.000,E1 42.732} C_DIS
LIN {X 0.128,Y -509.924,Z 847.035,A 0.000,B 0.000,C 90.000,E1 42.285} C_DIS
LIN {X -0.298,Y -504.774,Z 847.032,A 0.000,B 0.000,C 90.000,E1 41.757} C_DIS
LIN {X -0.172,Y -500.854,Z 847.029,A 0.000,B 0.000,C 90.000,E1 41.310} C_DIS
LIN {X -0.214,Y -493.987,Z 847.026,A 0.000,B 0.000,C 90.000,E1 40.620} C_DIS
LIN {X 0.078,Y -489.625,Z 847.023,A 0.000,B 0.000,C 90.000,E1 40.172} C_DIS
LIN {X 0.102,Y -483.760,Z 847.020,A 0.000,B 0.000,C 90.000,E1 39.644} C_DIS
LIN {X -0.172,Y -476.189,Z 847.017,A 0.000,B 0.000,C 90.000,E1 39.036} C_DIS
LIN {X 0.063,Y -468.405,Z 847.013,A 0.000,B 0.000,C 90.000,E1 38.382} C_DIS
LIN {X 0.178,Y -457.532,Z 847.009,A 0.000,B 0.000,C 90.000,E1 37.523} C_DIS
LIN {X -0.055,Y -449.578,Z 847.005,A 0.000,B 0.000,C 90.000,E1 36.950} C_DIS
LIN {X -0.164,Y -435.446,Z 846.999,A 0.000,B 0.000,C 90.000,E1 35.884} C_DIS
LIN {X 0.195,Y -415.466,Z 846.990,A 0.000,B 0.000,C 90.000,E1 34.199} C_DIS
LIN {X -0.213,Y -403.596,Z 846.984,A 0.000,B 0.000,C 90.000,E1 33.166} C_DIS
LIN {X -0.023,Y -398.213,Z 846.981,A 0.000,B 0.000,C 90.000,E1 32.546} C_DIS
LIN {X 0.025,Y -395.693,Z 846.979,A 0.000,B 0.000,C 90.000,E1 32.212} C_DIS
LIN {X 0.000,Y -394.805,Z 846.978,A 0.000,B 0.000,C 90.000,E1 32.084} C_DIS
LIN {X -0.090,Y -393.872,Z 846.977,A 0.000,B 0.000,C 90.000,E1 31.878} C_DIS
LIN {X -0.175,Y -390.638,Z 846.968,A 0.000,B 0.000,C 90.000,E1 30.207} C_DIS
LIN {X 0.061,Y -390.489,Z 846.964,A 0.000,B 0.000,C 90.000,E1 29.461} C_DIS
LIN {X -0.031,Y -392.873,Z 846.940,A 0.000,B 0.000,C 90.000,E1 25.207} C_DIS
LIN {X -0.121,Y -395.115,Z 846.924,A 0.000,B 0.000,C 90.000,E1 22.386} C_DIS
LIN {X 0.092,Y -397.301,Z 846.911,A 0.000,B 0.000,C 90.000,E1 19.885} C_DIS
LIN {X -0.133,Y -399.932,Z 846.897,A 0.000,B 0.000,C 90.000,E1 17.457} C_DIS
LIN {X 0.017,Y -404.363,Z 846.878,A 0.000,B 0.000,C 90.000,E1 13.939} C_DIS
LIN {X 0.212,Y -407.442,Z 846.866,A 0.000,B 0.000,C 90.000,E1 11.827} C_DIS
LIN {X -0.040,Y -411.322,Z 846.852,A 0.000,B 0.000,C 90.000,E1 9.443} C_DIS
LIN {X 0.170,Y -415.459,Z 846.839,A 0.000,B 0.000,C 90.000,E1 7.011} C_DIS
LIN {X 0.021,Y -419.770,Z 846.826,A 0.000,B 0.000,C 90.000,E1 4.645} C_DIS
LIN {X -0.003,Y -425.834,Z 846.809,A 0.000,B 0.000,C 90.000,E1 1.604} C_DIS
LIN {X -0.196,Y -430.611,Z 846.797,A 0.000,B 0.000,C 90.000,E1 359.484} C_DIS
LIN {X -0.039,Y -436.229,Z 846.784,A 0.000,B 0.000,C 90.000,E1 357.135} C_DIS
LIN {X 0.214,Y -441.122,Z 846.773,A 0.000,B 0.000,C 90.000,E1 355.122} C_DIS
LIN {X 0.150,Y -446.475,Z 846.762,A 0.000,B 0.000,C 90.000,E1 353.166} C_DIS
LIN {X -0.057,Y -448.220,Z 846.759,A 0.000,B 0.000,C 90.000,E1 352.704} C_DIS
LIN {X -0.185,Y -450.536,Z 846.757,A 0.000,B 0.000,C 90.000,E1 352.243} C_DIS
LIN {X 0.157,Y -452.919,Z 846.755,A 0.000,B 0.000,C 90.000,E1 351.837} C_DIS
LIN {X -0.034,Y -453.608,Z 846.754,A 0.000,B 0.000,C 90.000,E1 351.781} C_DIS
LIN {X -0.004,Y -457.724,Z 846.752,A 0.000,B 0.000,C 90.000,E1 351.432} C_DIS
LIN {X -0.093,Y -459.513,Z 846.752,A 0.000,B 0.000,C 90.000,E1 351.319} C_DIS
LIN {X 0.146,Y -464.942,Z 846.750,A 0.000,B 0.000,C 90.000,E1 350.971} C_DIS
LIN {X 0.005,Y -479.742,Z 846.746,A 0.000,B 0.000,C 90.000,E1 350.208} C_DIS
LIN {X 0.111,Y -489.441,Z 846.743,A 0.000,B 0.000,C 90.000,E1 349.634} C_DIS
LIN {X 0.234,Y -502.270,Z 846.738,A 0.000,B 0.000,C 90.000,E1 348.814} C_DIS
LIN {X 0.165,Y -508.569,Z 846.736,A 0.000,B 0.000,C 90.000,E1 348.409} C_DIS
LIN {X -0.139,Y -521.081,Z 846.731,A 0.000,B 0.000,C 90.000,E1 347.589} C_DIS
LIN {X -0.243,Y -530.093,Z 846.727,A 0.000,B 0.000,C 90.000,E1 346.937} C_DIS
LIN {X -0.134,Y -540.356,Z 846.723,A 0.000,B 0.000,C 90.000,E1 346.117} C_DIS
LIN {X -0.187,Y -546.121,Z 846.720,A 0.000,B 0.000,C 90.000,E1 345.644} C_DIS
LIN {X 0.142,Y -553.047,Z 846.717,A 0.000,B 0.000,C 90.000,E1 344.991} C_DIS
LIN {X -0.223,Y -559.730,Z 846.713,A 0.000,B 0.000,C 90.000,E1 344.393} C_DIS
LIN {X -0.188,Y -564.844,Z 846.710,A 0.000,B 0.000,C 90.000,E1 343.866} C_DIS
LIN {X -0.149,Y -569.758,Z 846.707,A 0.000,B 0.000,C 90.000,E1 343.323} C_DIS
LIN {X -0.001,Y -576.891,Z 846.703,A 0.000,B 0.000,C 90.000,E1 342.489} C_DIS
LIN {X -0.153,Y -583.247,Z 846.698,A 0.000,B 0.000,C 90.000,E1 341.692} C_DIS
LIN {X 0.133,Y -589.295,Z 846.694,A 0.000,B 0.000,C 90.000,E1 340.859} C_DIS
LIN {X 0.177,Y -593.773,Z 846.690,A 0.000,B 0.000,C 90.000,E1 340.188} C_DIS
LIN {X 0.118,Y -600.395,Z 846.684,A 0.000,B 0.000,C 90.000,E1 339.135} C_DIS
LIN {X -0.067,Y -606.587,Z 846.678,A 0.000,B 0.000,C 90.000,E1 338.103} C_DIS
LIN {X 0.070,Y -611.692,Z 846.673,A 0.000,B 0.000,C 90.000,E1 337.177} C_DIS
LIN {X -0.311,Y -617.274,Z 846.668,A 0.000,B 0.000,C 90.000,E1 336.177} C_DIS
LIN {X 0.203,Y -623.129,Z 846.661,A 0.000,B 0.000,C 90.000,E1 334.973} C_DIS
LIN {X -0.027,Y -628.577,Z 846.655,A 0.000,B 0.000,C 90.000,E1 333.845} C_DIS
LIN {X 0.039,Y -631.917,Z 846.651,A 0.000,B 0.000,C 90.000,E1 333.076} C_DIS
LIN {X -0.040,Y -637.158,Z 846.643,A 0.000,B 0.000,C 90.000,E1 331.820} C_DIS
LIN {X 0.171,Y -641.129,Z 846.638,A 0.000,B 0.000,C 90.000,E1 330.795} C_DIS
LIN {X 0.187,Y -644.975,Z 846.632,A 0.000,B 0.000,C 90.000,E1 329.793} C_DIS
LIN {X -0.136,Y -650.140,Z 846.624,A 0.000,B 0.000,C 90.000,E1 328.329} C_DIS
LIN {X 0.375,Y -651.726,Z 846.621,A 0.000,B 0.000,C 90.000,E1 327.788} C_DIS
LIN {X 0.069,Y -655.503,Z 846.614,A 0.000,B 0.000,C 90.000,E1 326.580} C_DIS
LIN {X -0.368,Y -658.931,Z 846.608,A 0.000,B 0.000,C 90.000,E1 325.388} C_DIS
LIN {X 0.135,Y -660.785,Z 846.604,A 0.000,B 0.000,C 90.000,E1 324.609} C_DIS
LIN {X 0.224,Y -663.048,Z 846.598,A 0.000,B 0.000,C 90.000,E1 323.623} C_DIS
LIN {X -0.098,Y -665.577,Z 846.591,A 0.000,B 0.000,C 90.000,E1 322.431} C_DIS
LIN {X 0.429,Y -667.669,Z 846.585,A 0.000,B 0.000,C 90.000,E1 321.170} C_DIS
LIN {X -0.021,Y -668.846,Z 846.581,A 0.000,B 0.000,C 90.000,E1 320.481} C_DIS
LIN {X 0.135,Y -670.517,Z 846.574,A 0.000,B 0.000,C 90.000,E1 319.256} C_DIS
LIN {X 0.297,Y -673.376,Z 846.562,A 0.000,B 0.000,C 90.000,E1 317.067} C_DIS
LIN {X -0.076,Y -674.702,Z 846.556,A 0.000,B 0.000,C 90.000,E1 316.134} C_DIS
LIN {X -0.023,Y -675.171,Z 846.554,A 0.000,B 0.000,C 90.000,E1 315.648} C_DIS
LIN {X 0.006,Y -675.573,Z 846.552,A 0.000,B 0.000,C 90.000,E1 315.405} C_DIS
LIN {X 0.262,Y -677.591,Z 846.542,A 0.000,B 0.000,C 90.000,E1 313.461} C_DIS
LIN {X -0.408,Y -679.323,Z 846.532,A 0.000,B 0.000,C 90.000,E1 311.838} C_DIS
LIN {X -0.196,Y -680.275,Z 846.527,A 0.000,B 0.000,C 90.000,E1 310.862} C_DIS
LIN {X 0.103,Y -681.576,Z 846.519,A 0.000,B 0.000,C 90.000,E1 309.402} C_DIS
LIN {X 0.090,Y -682.847,Z 846.511,A 0.000,B 0.000,C 90.000,E1 307.971} C_DIS
LIN {X 0.117,Y -684.048,Z 846.503,A 0.000,B 0.000,C 90.000,E1 306.537} C_DIS
LIN {X -0.021,Y -685.014,Z 846.496,A 0.000,B 0.000,C 90.000,E1 305.358} C_DIS
LIN {X 0.195,Y -685.980,Z 846.489,A 0.000,B 0.000,C 90.000,E1 303.913} C_DIS
LIN {X 0.270,Y -687.327,Z 846.478,A 0.000,B 0.000,C 90.000,E1 302.005} C_DIS
LIN {X 0.016,Y -688.715,Z 846.467,A 0.000,B 0.000,C 90.000,E1 300.129} C_DIS
LIN {X 0.189,Y -689.855,Z 846.460,A 0.000,B 0.000,C 90.000,E1 298.693} C_DIS
LIN {X 0.385,Y -691.072,Z 846.452,A 0.000,B 0.000,C 90.000,E1 297.257} C_DIS
LIN {X -0.096,Y -692.615,Z 846.442,A 0.000,B 0.000,C 90.000,E1 295.643} C_DIS
LIN {X -0.089,Y -693.675,Z 846.436,A 0.000,B 0.000,C 90.000,E1 294.463} C_DIS
LIN {X -0.266,Y -693.935,Z 846.432,A 0.000,B 0.000,C 90.000,E1 293.770} C_DIS
LIN {X 0.224,Y -693.722,Z 846.429,A 0.000,B 0.000,C 90.000,E1 293.259} C_DIS
LIN {X 0.196,Y -693.235,Z 846.428,A 0.000,B 0.000,C 90.000,E1 293.025} C_DIS
LIN {X -0.227,Y -691.406,Z 846.425,A 0.000,B 0.000,C 90.000,E1 292.589} C_DIS
LIN {X -0.108,Y -690.819,Z 846.425,A 0.000,B 0.000,C 90.000,E1 292.461} C_DIS
LIN {X 0.010,Y -689.932,Z 846.424,A 0.000,B 0.000,C 90.000,E1 292.333} C_DIS
LIN {X 0.177,Y -686.093,Z 846.422,A 0.000,B 0.000,C 90.000,E1 291.972} C_DIS
LIN {X -0.263,Y -684.675,Z 846.422,A 0.000,B 0.000,C 90.000,E1 291.897} C_DIS
LIN {X 0.001,Y -683.128,Z 846.421,A 0.000,B 0.000,C 90.000,E1 291.770} C_DIS
LIN {X 0.012,Y -680.747,Z 846.420,A 0.000,B 0.000,C 90.000,E1 291.663} C_DIS
LIN {X -0.047,Y -671.522,Z 846.419,A 0.000,B 0.000,C 90.000,E1 291.354} C_DIS
LIN {X 0.098,Y -663.477,Z 846.418,A 0.000,B 0.000,C 90.000,E1 291.153} C_DIS
LIN {X -0.275,Y -655.664,Z 846.417,A 0.000,B 0.000,C 90.000,E1 291.046} C_DIS
LIN {X 0.027,Y -648.598,Z 846.416,A 0.000,B 0.000,C 90.000,E1 290.844} C_DIS
LIN {X 0.065,Y -643.303,Z 846.415,A 0.000,B 0.000,C 90.000,E1 290.663} C_DIS
LIN {X 0.236,Y -638.078,Z 846.414,A 0.000,B 0.000,C 90.000,E1 290.429} C_DIS
LIN {X -0.128,Y -635.003,Z 846.412,A 0.000,B 0.000,C 90.000,E1 290.248} C_DIS
LIN {X -0.166,Y -634.989,Z 846.412,A 0.000,B 0.000,C 90.000,E1 290.248} C_DIS
LIN {X -0.161,Y -634.346,Z 846.411,A 0.000,B 0.000,C 90.000,E1 290.066} C_DIS
LIN {X -0.125,Y -635.473,Z 846.409,A 0.000,B 0.000,C 90.000,E1 289.685} C_DIS
LIN {X 0.190,Y -638.599,Z 846.406,A 0.000,B 0.000,C 90.000,E1 289.033} C_DIS
LIN {X 0.065,Y -642.164,Z 846.402,A 0.000,B 0.000,C 90.000,E1 288.417} C_DIS
LIN {X -0.175,Y -645.892,Z 846.398,A 0.000,B 0.000,C 90.000,E1 287.692} C_DIS
LIN {X 0.144,Y -648.170,Z 846.396,A 0.000,B 0.000,C 90.000,E1 287.166} C_DIS
LIN {X -0.085,Y -651.197,Z 846.391,A 0.000,B 0.000,C 90.000,E1 286.441} C_DIS
LIN {X 0.337,Y -653.809,Z 846.387,A 0.000,B 0.000,C 90.000,E1 285.662} C_DIS
LIN {X 0.095,Y -655.339,Z 846.384,A 0.000,B 0.000,C 90.000,E1 285.190} C_DIS
LIN {X -0.247,Y -657.102,Z 846.380,A 0.000,B 0.000,C 90.000,E1 284.481} C_DIS
LIN {X 0.067,Y -658.428,Z 846.376,A 0.000,B 0.000,C 90.000,E1 283.716} C_DIS
LIN {X -0.140,Y -659.054,Z 846.374,A 0.000,B 0.000,C 90.000,E1 283.244} C_DIS
LIN {X -0.346,Y -659.534,Z 846.371,A 0.000,B 0.000,C 90.000,E1 282.771} C_DIS
LIN {X 0.096,Y -659.770,Z 846.368,A 0.000,B 0.000,C 90.000,E1 282.243} C_DIS
LIN {X -0.211,Y -659.679,Z 846.364,A 0.000,B 0.000,C 90.000,E1 281.535} C_DIS
LIN {X 0.227,Y -659.405,Z 846.361,A 0.000,B 0.000,C 90.000,E1 281.007} C_DIS
LIN {X -0.108,Y -658.926,Z 846.359,A 0.000,B 0.000,C 90.000,E1 280.546} C_DIS
LIN {X 0.324,Y -658.229,Z 846.356,A 0.000,B 0.000,C 90.000,E1 280.018} C_DIS
LIN {X -0.128,Y -656.519,Z 846.352,A 0.000,B 0.000,C 90.000,E1 279.321} C_DIS
LIN {X 0.178,Y -655.022,Z 846.349,A 0.000,B 0.000,C 90.000,E1 278.803} C_DIS
LIN {X -0.169,Y -653.103,Z 846.346,A 0.000,B 0.000,C 90.000,E1 278.341} C_DIS
LIN {X 0.095,Y -650.210,Z 846.343,A 0.000,B 0.000,C 90.000,E1 277.701} C_DIS
LIN {X 0.243,Y -646.626,Z 846.339,A 0.000,B 0.000,C 90.000,E1 277.068} C_DIS
LIN {X -0.155,Y -643.478,Z 846.337,A 0.000,B 0.000,C 90.000,E1 276.606} C_DIS
LIN {X 0.066,Y -639.728,Z 846.334,A 0.000,B 0.000,C 90.000,E1 276.087} C_DIS
LIN {X -0.174,Y -634.296,Z 846.331,A 0.000,B 0.000,C 90.000,E1 275.511} C_DIS
LIN {X -0.261,Y -631.658,Z 846.329,A 0.000,B 0.000,C 90.000,E1 275.277} C_DIS
LIN {X -0.046,Y -627.935,Z 846.327,A 0.000,B 0.000,C 90.000,E1 274.935} C_DIS
LIN {X -0.033,Y -624.878,Z 846.326,A 0.000,B 0.000,C 90.000,E1 274.702} C_DIS
LIN {X -0.050,Y -618.896,Z 846.324,A 0.000,B 0.000,C 90.000,E1 274.302} C_DIS
LIN {X -0.148,Y -610.829,Z 846.321,A 0.000,B 0.000,C 90.000,E1 273.841} C_DIS
LIN {X 0.063,Y -600.625,Z 846.319,A 0.000,B 0.000,C 90.000,E1 273.326} C_DIS
LIN {X 0.248,Y -597.104,Z 846.318,A 0.000,B 0.000,C 90.000,E1 273.154} C_DIS
LIN {X -0.082,Y -590.339,Z 846.316,A 0.000,B 0.000,C 90.000,E1 272.922} C_DIS
LIN {X -0.226,Y -584.793,Z 846.315,A 0.000,B 0.000,C 90.000,E1 272.751} C_DIS
LIN {X -0.048,Y -578.443,Z 846.314,A 0.000,B 0.000,C 90.000,E1 272.579} C_DIS
LIN {X -0.254,Y -573.842,Z 846.314,A 0.000,B 0.000,C 90.000,E1 272.522} C_DIS
LIN {X 0.275,Y -568.532,Z 846.314,A 0.000,B 0.000,C 90.000,E1 272.407} C_DIS
LIN {X -0.081,Y -564.293,Z 846.313,A 0.000,B 0.000,C 90.000,E1 272.407} C_DIS
LIN {X -0.172,Y -558.934,Z 846.313,A 0.000,B 0.000,C 90.000,E1 272.407} C_DIS
LIN {X 0.054,Y -553.542,Z 846.313,A 0.000,B 0.000,C 90.000,E1 272.350} C_DIS
LIN {X 0.038,Y -550.227,Z 846.313,A 0.000,B 0.000,C 90.000,E1 272.236} C_DIS
LIN {X -0.002,Y -550.169,Z 846.312,A 0.000,B 0.000,C 90.000,E1 272.236} C_DIS
LIN {X -0.173,Y -549.086,Z 846.311,A 0.000,B 0.000,C 90.000,E1 272.064} C_DIS
LIN {X 0.198,Y -547.876,Z 846.309,A 0.000,B 0.000,C 90.000,E1 271.604} C_DIS
LIN {X -0.192,Y -546.973,Z 846.306,A 0.000,B 0.000,C 90.000,E1 271.088} C_DIS
LIN {X 0.218,Y -544.578,Z 846.290,A 0.000,B 0.000,C 90.000,E1 268.224} C_DIS
LIN {X -0.113,Y -543.610,Z 846.282,A 0.000,B 0.000,C 90.000,E1 266.846} C_DIS
LIN {X 0.120,Y -542.422,Z 846.273,A 0.000,B 0.000,C 90.000,E1 265.122} C_DIS
LIN {X -0.238,Y -541.442,Z 846.265,A 0.000,B 0.000,C 90.000,E1 263.742} C_DIS
LIN {X -0.089,Y -540.445,Z 846.259,A 0.000,B 0.000,C 90.000,E1 262.591} C_DIS
LIN {X 0.249,Y -538.907,Z 846.249,A 0.000,B 0.000,C 90.000,E1 260.849} C_DIS
LIN {X -0.102,Y -537.819,Z 846.243,A 0.000,B 0.000,C 90.000,E1 259.746} C_DIS
LIN {X 0.218,Y -536.389,Z 846.235,A 0.000,B 0.000,C 90.000,E1 258.285} C_DIS
LIN {X -0.071,Y -535.237,Z 846.229,A 0.000,B 0.000,C 90.000,E1 257.173} C_DIS
LIN {X 0.266,Y -533.906,Z 846.222,A 0.000,B 0.000,C 90.000,E1 255.992} C_DIS
LIN {X 0.145,Y -531.917,Z 846.213,A 0.000,B 0.000,C 90.000,E1 254.283} C_DIS
LIN {X 0.084,Y -530.214,Z 846.205,A 0.000,B 0.000,C 90.000,E1 252.851} C_DIS
LIN {X 0.150,Y -528.446,Z 846.197,A 0.000,B 0.000,C 90.000,E1 251.402} C_DIS
LIN {X -0.313,Y -526.585,Z 846.189,A 0.000,B 0.000,C 90.000,E1 250.007} C_DIS
LIN {X 0.030,Y -524.200,Z 846.179,A 0.000,B 0.000,C 90.000,E1 248.230} C_DIS
LIN {X -0.126,Y -522.125,Z 846.171,A 0.000,B 0.000,C 90.000,E1 246.794} C_DIS
LIN {X 0.010,Y -520.414,Z 846.165,A 0.000,B 0.000,C 90.000,E1 245.613} C_DIS
LIN {X 0.002,Y -518.070,Z 846.156,A 0.000,B 0.000,C 90.000,E1 244.152} C_DIS
LIN {X -0.156,Y -515.009,Z 846.147,A 0.000,B 0.000,C 90.000,E1 242.410} C_DIS
LIN {X 0.316,Y -511.880,Z 846.137,A 0.000,B 0.000,C 90.000,E1 240.589} C_DIS
LIN {X -0.153,Y -509.699,Z 846.130,A 0.000,B 0.000,C 90.000,E1 239.459} C_DIS
LIN {X 0.107,Y -506.924,Z 846.122,A 0.000,B 0.000,C 90.000,E1 237.946} C_DIS
LIN {X 0.213,Y -505.187,Z 846.117,A 0.000,B 0.000,C 90.000,E1 237.041} C_DIS
LIN {X -0.087,Y -502.628,Z 846.110,A 0.000,B 0.000,C 90.000,E1 235.881} C_DIS
LIN {X -0.141,Y -499.962,Z 846.104,A 0.000,B 0.000,C 90.000,E1 234.689} C_DIS
LIN {X 0.019,Y -498.498,Z 846.100,A 0.000,B 0.000,C 90.000,E1 234.069} C_DIS
LIN {X -0.059,Y -492.862,Z 846.087,A 0.000,B 0.000,C 90.000,E1 231.662} C_DIS
LIN {X 0.028,Y -488.613,Z 846.077,A 0.000,B 0.000,C 90.000,E1 229.828} C_DIS
LIN {X -0.187,Y -485.091,Z 846.068,A 0.000,B 0.000,C 90.000,E1 228.324} C_DIS
LIN {X 0.236,Y -479.620,Z 846.055,A 0.000,B 0.000,C 90.000,E1 225.810} C_DIS
LIN {X 0.154,Y -476.354,Z 846.046,A 0.000,B 0.000,C 90.000,E1 224.271} C_DIS
LIN {X -0.133,Y -471.569,Z 846.034,A 0.000,B 0.000,C 90.000,E1 222.123} C_DIS
LIN {X 0.003,Y -468.194,Z 846.025,A 0.000,B 0.000,C 90.000,E1 220.539} C_DIS
LIN {X 0.072,Y -464.938,Z 846.017,A 0.000,B 0.000,C 90.000,E1 218.955} C_DIS
LIN {X 0.112,Y -462.320,Z 846.009,A 0.000,B 0.000,C 90.000,E1 217.684} C_DIS
LIN {X -0.119,Y -458.357,Z 845.999,A 0.000,B 0.000,C 90.000,E1 215.804} C_DIS
LIN {X 0.033,Y -454.187,Z 845.988,A 0.000,B 0.000,C 90.000,E1 213.865} C_DIS
LIN {X 0.080,Y -450.055,Z 845.977,A 0.000,B 0.000,C 90.000,E1 211.926} C_DIS
LIN {X -0.137,Y -446.605,Z 845.969,A 0.000,B 0.000,C 90.000,E1 210.335} C_DIS
LIN {X 0.027,Y -442.662,Z 845.958,A 0.000,B 0.000,C 90.000,E1 208.359} C_DIS
LIN {X 0.110,Y -438.009,Z 845.945,A 0.000,B 0.000,C 90.000,E1 206.052} C_DIS
LIN {X 0.225,Y -434.653,Z 845.936,A 0.000,B 0.000,C 90.000,E1 204.387} C_DIS
LIN {X -0.089,Y -431.274,Z 845.926,A 0.000,B 0.000,C 90.000,E1 202.770} C_DIS
LIN {X 0.140,Y -427.367,Z 845.915,A 0.000,B 0.000,C 90.000,E1 200.737} C_DIS
LIN {X -0.091,Y -422.813,Z 845.902,A 0.000,B 0.000,C 90.000,E1 198.417} C_DIS
LIN {X -0.080,Y -418.901,Z 845.891,A 0.000,B 0.000,C 90.000,E1 196.386} C_DIS
LIN {X 0.047,Y -416.220,Z 845.883,A 0.000,B 0.000,C 90.000,E1 195.009} C_DIS
LIN {X 0.056,Y -412.732,Z 845.874,A 0.000,B 0.000,C 90.000,E1 193.300} C_DIS
LIN {X 0.016,Y -408.695,Z 845.863,A 0.000,B 0.000,C 90.000,E1 191.243} C_DIS
LIN {X 0.112,Y -405.401,Z 845.853,A 0.000,B 0.000,C 90.000,E1 189.500} C_DIS
LIN {X 0.140,Y -402.729,Z 845.845,A 0.000,B 0.000,C 90.000,E1 188.106} C_DIS
LIN {X -0.116,Y -396.748,Z 845.828,A 0.000,B 0.000,C 90.000,E1 184.992} C_DIS
LIN {X -0.194,Y -392.258,Z 845.812,A 0.000,B 0.000,C 90.000,E1 182.178} C_DIS
LIN {X -0.058,Y -388.293,Z 845.796,A 0.000,B 0.000,C 90.000,E1 179.312} C_DIS
LIN {X 0.051,Y -386.901,Z 845.790,A 0.000,B 0.000,C 90.000,E1 178.224} C_DIS
LIN {X 0.150,Y -383.504,Z 845.776,A 0.000,B 0.000,C 90.000,E1 175.698} C_DIS
LIN {X -0.101,Y -380.747,Z 845.764,A 0.000,B 0.000,C 90.000,E1 173.571} C_DIS
LIN {X -0.058,Y -377.767,Z 845.750,A 0.000,B 0.000,C 90.000,E1 171.027} C_DIS
LIN {X 0.129,Y -375.536,Z 845.738,A 0.000,B 0.000,C 90.000,E1 168.814} C_DIS
LIN {X -0.063,Y -373.440,Z 845.724,A 0.000,B 0.000,C 90.000,E1 166.284} C_DIS
LIN {X 0.036,Y -371.782,Z 845.703,A 0.000,B 0.000,C 90.000,E1 162.598} C_DIS
LIN {X -0.096,Y -372.239,Z 845.695,A 0.000,B 0.000,C 90.000,E1 161.148} C_DIS
LIN {X 0.159,Y -372.915,Z 845.689,A 0.000,B 0.000,C 90.000,E1 160.007} C_DIS
LIN {X 0.126,Y -373.222,Z 845.687,A 0.000,B 0.000,C 90.000,E1 159.645} C_DIS
LIN {X -0.153,Y -374.238,Z 845.683,A 0.000,B 0.000,C 90.000,E1 158.954} C_DIS
LIN {X -0.071,Y -375.596,Z 845.679,A 0.000,B 0.000,C 90.000,E1 158.209} C_DIS
LIN {X -0.120,Y -377.448,Z 845.675,A 0.000,B 0.000,C 90.000,E1 157.486} C_DIS
LIN {X 0.004,Y -378.608,Z 845.673,A 0.000,B 0.000,C 90.000,E1 157.102} C_DIS
LIN {X -0.005,Y -379.381,Z 845.672,A 0.000,B 0.000,C 90.000,E1 156.922} C_DIS
LIN {X -0.164,Y -382.045,Z 845.669,A 0.000,B 0.000,C 90.000,E1 156.485} C_DIS
LIN {X -0.018,Y -383.795,Z 845.667,A 0.000,B 0.000,C 90.000,E1 156.102} C_DIS
LIN {X -0.043,Y -385.485,Z 845.666,A 0.000,B 0.000,C 90.000,E1 155.845} C_DIS
LIN {X -0.041,Y -387.075,Z 845.665,A 0.000,B 0.000,C 90.000,E1 155.665} C_DIS
LIN {X 0.193,Y -391.883,Z 845.663,A 0.000,B 0.000,C 90.000,E1 155.229} C_DIS
LIN {X -0.098,Y -398.231,Z 845.661,A 0.000,B 0.000,C 90.000,E1 154.921} C_DIS
LIN {X 0.207,Y -402.077,Z 845.660,A 0.000,B 0.000,C 90.000,E1 154.717} C_DIS
LIN {X 0.083,Y -407.547,Z 845.659,A 0.000,B 0.000,C 90.000,E1 154.537} C_DIS
LIN {X 0.095,Y -421.180,Z 845.656,A 0.000,B 0.000,C 90.000,E1 153.973} C_DIS
LIN {X 0.124,Y -427.513,Z 845.654,A 0.000,B 0.000,C 90.000,E1 153.640} C_DIS
LIN {X -0.094,Y -435.658,Z 845.651,A 0.000,B 0.000,C 90.000,E1 153.204} C_DIS
LIN {X 0.032,Y -443.612,Z 845.648,A 0.000,B 0.000,C 90.000,E1 152.666} C_DIS
LIN {X -0.093,Y -450.047,Z 845.646,A 0.000,B 0.000,C 90.000,E1 152.231} C_DIS
LIN {X 0.135,Y -456.048,Z 845.643,A 0.000,B 0.000,C 90.000,E1 151.719} C_DIS
LIN {X 0.236,Y -463.281,Z 845.639,A 0.000,B 0.000,C 90.000,E1 151.051} C_DIS
LIN {X 0.020,Y -467.554,Z 845.637,A 0.000,B 0.000,C 90.000,E1 150.667} C_DIS
LIN {X 0.116,Y -473.082,Z 845.634,A 0.000,B 0.000,C 90.000,E1 150.078} C_DIS
LIN {X -0.190,Y -477.121,Z 845.631,A 0.000,B 0.000,C 90.000,E1 149.665} C_DIS
LIN {X 0.049,Y -481.384,Z 845.629,A 0.000,B 0.000,C 90.000,E1 149.203} C_DIS
LIN {X 0.044,Y -490.444,Z 845.623,A 0.000,B 0.000,C 90.000,E1 148.152} C_DIS
LIN {X 0.167,Y -495.272,Z 845.620,A 0.000,B 0.000,C 90.000,E1 147.533} C_DIS
LIN {X 0.037,Y -504.182,Z 845.613,A 0.000,B 0.000,C 90.000,E1 146.342} C_DIS
LIN {X 0.342,Y -506.392,Z 845.611,A 0.000,B 0.000,C 90.000,E1 146.008} C_DIS
LIN {X 0.086,Y -513.751,Z 845.605,A 0.000,B 0.000,C 90.000,E1 144.848} C_DIS
LIN {X -0.069,Y -521.481,Z 845.597,A 0.000,B 0.000,C 90.000,E1 143.543} C_DIS
LIN {X 0.334,Y -529.060,Z 845.590,A 0.000,B 0.000,C 90.000,E1 142.190} C_DIS
LIN {X 0.035,Y -539.758,Z 845.580,A 0.000,B 0.000,C 90.000,E1 140.356} C_DIS
LIN {X -0.110,Y -546.719,Z 845.573,A 0.000,B 0.000,C 90.000,E1 139.094} C_DIS
LIN {X 0.286,Y -556.360,Z 845.563,A 0.000,B 0.000,C 90.000,E1 137.229} C_DIS
LIN {X -0.200,Y -563.659,Z 845.555,A 0.000,B 0.000,C 90.000,E1 135.891} C_DIS
LIN {X -0.112,Y -568.418,Z 845.550,A 0.000,B 0.000,C 90.000,E1 134.919} C_DIS
LIN {X -0.001,Y -575.009,Z 845.542,A 0.000,B 0.000,C 90.000,E1 133.542} C_DIS
LIN {X -0.178,Y -581.435,Z 845.534,A 0.000,B 0.000,C 90.000,E1 132.204} C_DIS
LIN {X -0.105,Y -586.721,Z 845.528,A 0.000,B 0.000,C 90.000,E1 130.987} C_DIS
LIN {X -0.039,Y -592.400,Z 845.520,A 0.000,B 0.000,C 90.000,E1 129.644} C_DIS
LIN {X -0.103,Y -596.655,Z 845.514,A 0.000,B 0.000,C 90.000,E1 128.588} C_DIS
LIN {X -0.014,Y -600.332,Z 845.508,A 0.000,B 0.000,C 90.000,E1 127.523} C_DIS
LIN {X 0.137,Y -603.552,Z 845.503,A 0.000,B 0.000,C 90.000,E1 126.457} C_DIS
LIN {X -0.160,Y -606.399,Z 845.497,A 0.000,B 0.000,C 90.000,E1 125.438} C_DIS
LIN {X 0.023,Y -607.760,Z 845.494,A 0.000,B 0.000,C 90.000,E1 124.898} C_DIS
LIN {X -0.074,Y -609.910,Z 845.488,A 0.000,B 0.000,C 90.000,E1 123.865} C_DIS
LIN {X -0.088,Y -611.294,Z 845.484,A 0.000,B 0.000,C 90.000,E1 123.086} C_DIS
LIN {X -0.146,Y -612.842,Z 845.478,A 0.000,B 0.000,C 90.000,E1 122.054} C_DIS
LIN {X 0.014,Y -614.285,Z 845.472,A 0.000,B 0.000,C 90.000,E1 121.003} C_DIS
LIN {X -0.326,Y -615.506,Z 845.467,A 0.000,B 0.000,C 90.000,E1 120.001} C_DIS
LIN {X -0.073,Y -616.005,Z 845.464,A 0.000,B 0.000,C 90.000,E1 119.461} C_DIS
LIN {X 0.115,Y -616.875,Z 845.457,A 0.000,B 0.000,C 90.000,E1 118.153} C_DIS
LIN {X 0.080,Y -617.001,Z 845.454,A 0.000,B 0.000,C 90.000,E1 117.641} C_DIS
LIN {X 0.030,Y -616.805,Z 845.449,A 0.000,B 0.000,C 90.000,E1 116.873} C_DIS
LIN {X -0.037,Y -616.177,Z 845.444,A 0.000,B 0.000,C 90.000,E1 115.848} C_DIS
LIN {X -0.097,Y -615.511,Z 845.439,A 0.000,B 0.000,C 90.000,E1 115.079} C_DIS
LIN {X 0.139,Y -614.151,Z 845.435,A 0.000,B 0.000,C 90.000,E1 114.283} C_DIS
LIN {X 0.086,Y -613.014,Z 845.432,A 0.000,B 0.000,C 90.000,E1 113.770} C_DIS
LIN {X 0.022,Y -611.542,Z 845.429,A 0.000,B 0.000,C 90.000,E1 113.259} C_DIS
LIN {X -0.293,Y -609.627,Z 845.426,A 0.000,B 0.000,C 90.000,E1 112.770} C_DIS
LIN {X 0.226,Y -608.111,Z 845.425,A 0.000,B 0.000,C 90.000,E1 112.461} C_DIS
LIN {X 0.175,Y -606.320,Z 845.424,A 0.000,B 0.000,C 90.000,E1 112.206} C_DIS
LIN {X 0.146,Y -605.292,Z 845.423,A 0.000,B 0.000,C 90.000,E1 112.078} C_DIS
LIN {X -0.136,Y -601.638,Z 845.421,A 0.000,B 0.000,C 90.000,E1 111.716} C_DIS
LIN {X -0.297,Y -599.531,Z 845.420,A 0.000,B 0.000,C 90.000,E1 111.535} C_DIS
LIN {X -0.014,Y -594.915,Z 845.418,A 0.000,B 0.000,C 90.000,E1 111.153} C_DIS
LIN {X 0.159,Y -588.313,Z 845.415,A 0.000,B 0.000,C 90.000,E1 110.737} C_DIS
LIN {X 0.144,Y -584.800,Z 845.414,A 0.000,B 0.000,C 90.000,E1 110.556} C_DIS
LIN {X 0.273,Y -579.513,Z 845.413,A 0.000,B 0.000,C 90.000,E1 110.301} C_DIS
LIN {X -0.071,Y -571.427,Z 845.411,A 0.000,B 0.000,C 90.000,E1 109.993} C_DIS
LIN {X -0.269,Y -570.080,Z 845.411,A 0.000,B 0.000,C 90.000,E1 109.939} C_DIS
LIN {X -0.266,Y -565.169,Z 845.409,A 0.000,B 0.000,C 90.000,E1 109.577} C_DIS
LIN {X -0.300,Y -565.142,Z 845.409,A 0.000,B 0.000,C 90.000,E1 109.577} C_DIS
LIN {X -0.063,Y -564.322,Z 845.408,A 0.000,B 0.000,C 90.000,E1 109.396} C_DIS
LIN {X -0.132,Y -562.574,Z 845.405,A 0.000,B 0.000,C 90.000,E1 108.852} C_DIS
LIN {X 0.145,Y -561.509,Z 845.401,A 0.000,B 0.000,C 90.000,E1 108.127} C_DIS
LIN {X 0.056,Y -561.115,Z 845.398,A 0.000,B 0.000,C 90.000,E1 107.583} C_DIS
LIN {X -0.092,Y -560.944,Z 845.387,A 0.000,B 0.000,C 90.000,E1 105.662} C_DIS
LIN {X 0.046,Y -562.017,Z 845.372,A 0.000,B 0.000,C 90.000,E1 102.883} C_DIS
LIN {X -0.192,Y -563.568,Z 845.358,A 0.000,B 0.000,C 90.000,E1 100.423} C_DIS
LIN {X 0.035,Y -564.757,Z 845.349,A 0.000,B 0.000,C 90.000,E1 98.746} C_DIS
LIN {X 0.212,Y -565.685,Z 845.341,A 0.000,B 0.000,C 90.000,E1 97.352} C_DIS
LIN {X -0.140,Y -566.624,Z 845.332,A 0.000,B 0.000,C 90.000,E1 95.739} C_DIS
LIN {X -0.068,Y -567.238,Z 845.324,A 0.000,B 0.000,C 90.000,E1 94.359} C_DIS
LIN {X -0.138,Y -567.679,Z 845.318,A 0.000,B 0.000,C 90.000,E1 93.269} C_DIS
LIN {X -0.078,Y -568.107,Z 845.311,A 0.000,B 0.000,C 90.000,E1 91.892} C_DIS
LIN {X 0.108,Y -568.549,Z 845.301,A 0.000,B 0.000,C 90.000,E1 90.229} C_DIS
LIN {X -0.156,Y -569.036,Z 845.291,A 0.000,B 0.000,C 90.000,E1 88.339} C_DIS
LIN {X -0.085,Y -569.297,Z 845.283,A 0.000,B 0.000,C 90.000,E1 86.963} C_DIS
LIN {X 0.148,Y -569.539,Z 845.274,A 0.000,B 0.000,C 90.000,E1 85.298} C_DIS
LIN {X -0.244,Y -569.834,Z 845.266,A 0.000,B 0.000,C 90.000,E1 83.970} C_DIS
LIN {X -0.223,Y -570.320,Z 845.254,A 0.000,B 0.000,C 90.000,E1 81.781} C_DIS
LIN {X -0.133,Y -570.862,Z 845.244,A 0.000,B 0.000,C 90.000,E1 79.859} C_DIS
LIN {X -0.215,Y -571.458,Z 845.235,A 0.000,B 0.000,C 90.000,E1 78.229} C_DIS
LIN {X -0.006,Y -571.826,Z 845.228,A 0.000,B 0.000,C 90.000,E1 77.117} C_DIS
LIN {X 0.168,Y -572.301,Z 845.219,A 0.000,B 0.000,C 90.000,E1 75.463} C_DIS
LIN {X 0.157,Y -572.511,Z 845.212,A 0.000,B 0.000,C 90.000,E1 74.102} C_DIS
LIN {X -0.241,Y -572.690,Z 845.204,A 0.000,B 0.000,C 90.000,E1 72.779} C_DIS
LIN {X 0.266,Y -572.716,Z 845.195,A 0.000,B 0.000,C 90.000,E1 71.094} C_DIS
LIN {X -0.317,Y -572.609,Z 845.186,A 0.000,B 0.000,C 90.000,E1 69.518} C_DIS
LIN {X -0.132,Y -572.388,Z 845.175,A 0.000,B 0.000,C 90.000,E1 67.592} C_DIS
LIN {X 0.220,Y -572.102,Z 845.166,A 0.000,B 0.000,C 90.000,E1 65.921} C_DIS
LIN {X -0.085,Y -571.640,Z 845.159,A 0.000,B 0.000,C 90.000,E1 64.588} C_DIS
LIN {X -0.056,Y -571.002,Z 845.150,A 0.000,B 0.000,C 90.000,E1 62.948} C_DIS
LIN {X 0.039,Y -570.641,Z 845.144,A 0.000,B 0.000,C 90.000,E1 61.847} C_DIS
LIN {X 0.126,Y -570.062,Z 845.138,A 0.000,B 0.000,C 90.000,E1 60.745} C_DIS
LIN {X -0.008,Y -569.270,Z 845.132,A 0.000,B 0.000,C 90.000,E1 59.665} C_DIS
LIN {X -0.142,Y -568.199,Z 845.125,A 0.000,B 0.000,C 90.000,E1 58.584} C_DIS
LIN {X 0.190,Y -567.037,Z 845.119,A 0.000,B 0.000,C 90.000,E1 57.454} C_DIS
LIN {X 0.019,Y -565.634,Z 845.113,A 0.000,B 0.000,C 90.000,E1 56.373} C_DIS
LIN {X 0.031,Y -564.451,Z 845.109,A 0.000,B 0.000,C 90.000,E1 55.548} C_DIS
LIN {X 0.352,Y -563.149,Z 845.104,A 0.000,B 0.000,C 90.000,E1 54.689} C_DIS
LIN {X -0.020,Y -561.104,Z 845.098,A 0.000,B 0.000,C 90.000,E1 53.623} C_DIS
LIN {X 0.272,Y -559.405,Z 845.093,A 0.000,B 0.000,C 90.000,E1 52.763} C_DIS
LIN {X -0.155,Y -556.806,Z 845.087,A 0.000,B 0.000,C 90.000,E1 51.698} C_DIS
LIN {X 0.005,Y -555.347,Z 845.084,A 0.000,B 0.000,C 90.000,E1 51.126} C_DIS
LIN {X 0.075,Y -553.795,Z 845.081,A 0.000,B 0.000,C 90.000,E1 50.561} C_DIS
LIN {X -0.150,Y -551.155,Z 845.076,A 0.000,B 0.000,C 90.000,E1 49.747} C_DIS
LIN {X -0.041,Y -548.082,Z 845.072,A 0.000,B 0.000,C 90.000,E1 48.895} C_DIS
LIN {X 0.045,Y -545.921,Z 845.069,A 0.000,B 0.000,C 90.000,E1 48.324} C_DIS
LIN {X -0.101,Y -542.978,Z 845.065,A 0.000,B 0.000,C 90.000,E1 47.634} C_DIS
LIN {X 0.092,Y -539.696,Z 845.061,A 0.000,B 0.000,C 90.000,E1 46.905} C_DIS
LIN {X -0.297,Y -536.904,Z 845.058,A 0.000,B 0.000,C 90.000,E1 46.377} C_DIS
LIN {X -0.334,Y -533.817,Z 845.054,A 0.000,B 0.000,C 90.000,E1 45.810} C_DIS
LIN {X -0.222,Y -529.464,Z 845.050,A 0.000,B 0.000,C 90.000,E1 45.081} C_DIS
LIN {X -0.149,Y -524.632,Z 845.046,A 0.000,B 0.000,C 90.000,E1 44.352} C_DIS
LIN {X 0.313,Y -521.584,Z 845.044,A 0.000,B 0.000,C 90.000,E1 43.866} C_DIS
LIN {X -0.050,Y -515.984,Z 845.040,A 0.000,B 0.000,C 90.000,E1 43.176} C_DIS
LIN {X -0.020,Y -512.428,Z 845.037,A 0.000,B 0.000,C 90.000,E1 42.732} C_DIS
LIN {X 0.017,Y -508.664,Z 845.035,A 0.000,B 0.000,C 90.000,E1 42.285} C_DIS
LIN {X 0.222,Y -503.355,Z 845.032,A 0.000,B 0.000,C 90.000,E1 41.676} C_DIS
LIN {X -0.163,Y -499.509,Z 845.029,A 0.000,B 0.000,C 90.000,E1 41.310} C_DIS
LIN {X 0.032,Y -494.087,Z 845.026,A 0.000,B 0.000,C 90.000,E1 40.744} C_DIS
LIN {X 0.000,Y -489.777,Z 845.024,A 0.000,B 0.000,C 90.000,E1 40.334} C_DIS
LIN {X 0.281,Y -482.280,Z 845.021,A 0.000,B 0.000,C 90.000,E1 39.644} C_DIS
LIN {X 0.075,Y -474.721,Z 845.017,A 0.000,B 0.000,C 90.000,E1 39.036} C_DIS
LIN {X -0.300,Y -466.900,Z 845.014,A 0.000,B 0.000,C 90.000,E1 38.463} C_DIS
LIN {X 0.144,Y -454.384,Z 845.008,A 0.000,B 0.000,C 90.000,E1 37.443} C_DIS
LIN {X 0.038,Y -437.001,Z 845.001,A 0.000,B 0.000,C 90.000,E1 36.137} C_DIS
LIN {X -0.130,Y -415.467,Z 844.991,A 0.000,B 0.000,C 90.000,E1 34.405} C_DIS
LIN {X 0.104,Y -405.035,Z 844.986,A 0.000,B 0.000,C 90.000,E1 33.420} C_DIS
LIN {X -0.004,Y -400.836,Z 844.983,A 0.000,B 0.000,C 90.000,E1 33.007} C_DIS
LIN {X -0.203,Y -397.298,Z 844.981,A 0.000,B 0.000,C 90.000,E1 32.625} C_DIS
LIN {X 0.042,Y -394.383,Z 844.979,A 0.000,B 0.000,C 90.000,E1 32.163} C_DIS
LIN {X -0.113,Y -394.008,Z 844.978,A 0.000,B 0.000,C 90.000,E1 32.005} C_DIS
LIN {X 0.155,Y -392.708,Z 844.974,A 0.000,B 0.000,C 90.000,E1 31.258} C_DIS
LIN {X 0.068,Y -390.702,Z 844.968,A 0.000,B 0.000,C 90.000,E1 30.207} C_DIS
LIN {X -0.036,Y -390.732,Z 844.962,A 0.000,B 0.000,C 90.000,E1 29.155} C_DIS
LIN {X 0.021,Y -392.779,Z 844.942,A 0.000,B 0.000,C 90.000,E1 25.591} C_DIS
LIN {X -0.116,Y -394.648,Z 844.928,A 0.000,B 0.000,C 90.000,E1 23.131} C_DIS
LIN {X 0.156,Y -396.470,Z 844.917,A 0.000,B 0.000,C 90.000,E1 20.972} C_DIS
LIN {X 0.058,Y -399.636,Z 844.899,A 0.000,B 0.000,C 90.000,E1 17.819} C_DIS
LIN {X -0.027,Y -401.676,Z 844.889,A 0.000,B 0.000,C 90.000,E1 16.079} C_DIS
LIN {X -0.102,Y -404.954,Z 844.876,A 0.000,B 0.000,C 90.000,E1 13.647} C_DIS
LIN {X 0.110,Y -408.069,Z 844.864,A 0.000,B 0.000,C 90.000,E1 11.535} C_DIS
LIN {X -0.127,Y -412.009,Z 844.851,A 0.000,B 0.000,C 90.000,E1 9.151} C_DIS
LIN {X 0.061,Y -414.957,Z 844.841,A 0.000,B 0.000,C 90.000,E1 7.409} C_DIS
LIN {X -0.165,Y -418.650,Z 844.830,A 0.000,B 0.000,C 90.000,E1 5.391} C_DIS
LIN {X 0.194,Y -424.515,Z 844.813,A 0.000,B 0.000,C 90.000,E1 2.293} C_DIS
LIN {X 0.163,Y -430.063,Z 844.799,A 0.000,B 0.000,C 90.000,E1 359.771} C_DIS
LIN {X -0.032,Y -436.402,Z 844.784,A 0.000,B 0.000,C 90.000,E1 357.135} C_DIS
LIN {X 0.225,Y -441.287,Z 844.773,A 0.000,B 0.000,C 90.000,E1 355.122} C_DIS
LIN {X 0.164,Y -446.545,Z 844.762,A 0.000,B 0.000,C 90.000,E1 353.166} C_DIS
LIN {X -0.043,Y -448.174,Z 844.759,A 0.000,B 0.000,C 90.000,E1 352.704} C_DIS
LIN {X 0.023,Y -450.699,Z 844.756,A 0.000,B 0.000,C 90.000,E1 352.129} C_DIS
LIN {X -0.182,Y -453.086,Z 844.754,A 0.000,B 0.000,C 90.000,E1 351.781} C_DIS
LIN {X 0.142,Y -453.723,Z 844.754,A 0.000,B 0.000,C 90.000,E1 351.659} C_DIS
LIN {X -0.190,Y -459.666,Z 844.751,A 0.000,B 0.000,C 90.000,E1 351.197} C_DIS
LIN {X -0.114,Y -465.447,Z 844.749,A 0.000,B 0.000,C 90.000,E1 350.849} C_DIS
LIN {X 0.114,Y -473.428,Z 844.747,A 0.000,B 0.000,C 90.000,E1 350.387} C_DIS
LIN {X -0.128,Y -478.487,Z 844.745,A 0.000,B 0.000,C 90.000,E1 350.151} C_DIS
LIN {X 0.080,Y -488.147,Z 844.742,A 0.000,B 0.000,C 90.000,E1 349.567} C_DIS
LIN {X 0.068,Y -499.443,Z 844.738,A 0.000,B 0.000,C 90.000,E1 348.870} C_DIS
LIN {X 0.239,Y -507.273,Z 844.735,A 0.000,B 0.000,C 90.000,E1 348.342} C_DIS
LIN {X 0.059,Y -521.192,Z 844.730,A 0.000,B 0.000,C 90.000,E1 347.409} C_DIS
LIN {X -0.062,Y -530.226,Z 844.726,A 0.000,B 0.000,C 90.000,E1 346.756} C_DIS
LIN {X 0.059,Y -540.580,Z 844.722,A 0.000,B 0.000,C 90.000,E1 345.936} C_DIS
LIN {X 0.101,Y -547.648,Z 844.719,A 0.000,B 0.000,C 90.000,E1 345.338} C_DIS
LIN {X -0.075,Y -553.154,Z 844.716,A 0.000,B 0.000,C 90.000,E1 344.866} C_DIS
LIN {X 0.153,Y -559.766,Z 844.712,A 0.000,B 0.000,C 90.000,E1 344.212} C_DIS
LIN {X 0.211,Y -564.905,Z 844.710,A 0.000,B 0.000,C 90.000,E1 343.685} C_DIS
LIN {X 0.255,Y -569.845,Z 844.707,A 0.000,B 0.000,C 90.000,E1 343.142} C_DIS
LIN {X -0.140,Y -576.970,Z 844.702,A 0.000,B 0.000,C 90.000,E1 342.362} C_DIS
LIN {X -0.207,Y -582.309,Z 844.698,A 0.000,B 0.000,C 90.000,E1 341.692} C_DIS
LIN {X -0.002,Y -589.427,Z 844.693,A 0.000,B 0.000,C 90.000,E1 340.732} C_DIS
LIN {X 0.044,Y -593.883,Z 844.689,A 0.000,B 0.000,C 90.000,E1 340.061} C_DIS
LIN {X -0.226,Y -600.509,Z 844.683,A 0.000,B 0.000,C 90.000,E1 339.028} C_DIS
LIN {X -0.163,Y -605.942,Z 844.678,A 0.000,B 0.000,C 90.000,E1 338.103} C_DIS
LIN {X -0.056,Y -611.814,Z 844.673,A 0.000,B 0.000,C 90.000,E1 337.050} C_DIS
LIN {X 0.142,Y -616.713,Z 844.667,A 0.000,B 0.000,C 90.000,E1 336.125} C_DIS
LIN {X 0.080,Y -622.626,Z 844.661,A 0.000,B 0.000,C 90.000,E1 334.973} C_DIS
LIN {X 0.111,Y -627.543,Z 844.655,A 0.000,B 0.000,C 90.000,E1 333.948} C_DIS
LIN {X -0.108,Y -630.935,Z 844.651,A 0.000,B 0.000,C 90.000,E1 333.204} C_DIS
LIN {X 0.357,Y -636.274,Z 844.644,A 0.000,B 0.000,C 90.000,E1 331.897} C_DIS
LIN {X -0.004,Y -640.320,Z 844.638,A 0.000,B 0.000,C 90.000,E1 330.923} C_DIS
LIN {X 0.000,Y -644.213,Z 844.633,A 0.000,B 0.000,C 90.000,E1 329.921} C_DIS
LIN {X -0.345,Y -646.896,Z 844.629,A 0.000,B 0.000,C 90.000,E1 329.203} C_DIS
LIN {X -0.255,Y -650.336,Z 844.623,A 0.000,B 0.000,C 90.000,E1 328.201} C_DIS
LIN {X -0.141,Y -655.020,Z 844.615,A 0.000,B 0.000,C 90.000,E1 326.707} C_DIS
LIN {X -0.135,Y -657.805,Z 844.610,A 0.000,B 0.000,C 90.000,E1 325.722} C_DIS
LIN {X -0.083,Y -660.446,Z 844.604,A 0.000,B 0.000,C 90.000,E1 324.736} C_DIS
LIN {X 0.102,Y -663.294,Z 844.597,A 0.000,B 0.000,C 90.000,E1 323.497} C_DIS
LIN {X -0.315,Y -665.297,Z 844.592,A 0.000,B 0.000,C 90.000,E1 322.557} C_DIS
LIN {X 0.229,Y -667.107,Z 844.586,A 0.000,B 0.000,C 90.000,E1 321.537} C_DIS
LIN {X -0.144,Y -668.727,Z 844.581,A 0.000,B 0.000,C 90.000,E1 320.598} C_DIS
LIN {X -0.068,Y -670.774,Z 844.573,A 0.000,B 0.000,C 90.000,E1 319.138} C_DIS
LIN {X -0.357,Y -673.395,Z 844.562,A 0.000,B 0.000,C 90.000,E1 317.229} C_DIS
LIN {X 0.176,Y -674.091,Z 844.560,A 0.000,B 0.000,C 90.000,E1 316.701} C_DIS
LIN {X 0.249,Y -675.012,Z 844.556,A 0.000,B 0.000,C 90.000,E1 315.972} C_DIS
LIN {X -0.053,Y -676.626,Z 844.548,A 0.000,B 0.000,C 90.000,E1 314.555} C_DIS
LIN {X 0.170,Y -678.179,Z 844.540,A 0.000,B 0.000,C 90.000,E1 313.095} C_DIS
LIN {X -0.028,Y -679.946,Z 844.530,A 0.000,B 0.000,C 90.000,E1 311.434} C_DIS
LIN {X -0.178,Y -681.295,Z 844.522,A 0.000,B 0.000,C 90.000,E1 310.011} C_DIS
LIN {X 0.228,Y -682.562,Z 844.514,A 0.000,B 0.000,C 90.000,E1 308.543} C_DIS
LIN {X 0.086,Y -683.592,Z 844.508,A 0.000,B 0.000,C 90.000,E1 307.363} C_DIS
LIN {X 0.090,Y -684.584,Z 844.501,A 0.000,B 0.000,C 90.000,E1 306.171} C_DIS
LIN {X 0.121,Y -685.511,Z 844.494,A 0.000,B 0.000,C 90.000,E1 304.978} C_DIS
LIN {X -0.209,Y -686.475,Z 844.487,A 0.000,B 0.000,C 90.000,E1 303.579} C_DIS
LIN {X 0.254,Y -687.669,Z 844.477,A 0.000,B 0.000,C 90.000,E1 301.878} C_DIS
LIN {X -0.213,Y -688.897,Z 844.468,A 0.000,B 0.000,C 90.000,E1 300.256} C_DIS
LIN {X 0.194,Y -690.202,Z 844.459,A 0.000,B 0.000,C 90.000,E1 298.565} C_DIS
LIN {X -0.217,Y -691.416,Z 844.451,A 0.000,B 0.000,C 90.000,E1 297.180} C_DIS
LIN {X -0.078,Y -692.945,Z 844.442,A 0.000,B 0.000,C 90.000,E1 295.515} C_DIS
LIN {X -0.312,Y -693.770,Z 844.437,A 0.000,B 0.000,C 90.000,E1 294.591} C_DIS
LIN {X 0.428,Y -694.122,Z 844.433,A 0.000,B 0.000,C 90.000,E1 293.823} C_DIS
LIN {X 0.005,Y -693.904,Z 844.430,A 0.000,B 0.000,C 90.000,E1 293.387} C_DIS
LIN {X -0.024,Y -693.694,Z 844.429,A 0.000,B 0.000,C 90.000,E1 293.153} C_DIS
LIN {X 0.221,Y -692.899,Z 844.427,A 0.000,B 0.000,C 90.000,E1 292.898} C_DIS
LIN {X -0.203,Y -690.806,Z 844.425,A 0.000,B 0.000,C 90.000,E1 292.461} C_DIS
LIN {X -0.086,Y -689.897,Z 844.424,A 0.000,B 0.000,C 90.000,E1 292.333} C_DIS
LIN {X 0.193,Y -687.320,Z 844.423,A 0.000,B 0.000,C 90.000,E1 292.078} C_DIS
LIN {X 0.047,Y -682.831,Z 844.421,A 0.000,B 0.000,C 90.000,E1 291.770} C_DIS
LIN {X 0.159,Y -680.636,Z 844.420,A 0.000,B 0.000,C 90.000,E1 291.663} C_DIS
LIN {X -0.053,Y -670.886,Z 844.419,A 0.000,B 0.000,C 90.000,E1 291.354} C_DIS
LIN {X -0.341,Y -663.931,Z 844.418,A 0.000,B 0.000,C 90.000,E1 291.227} C_DIS
LIN {X -0.230,Y -654.555,Z 844.417,A 0.000,B 0.000,C 90.000,E1 291.046} C_DIS
LIN {X 0.015,Y -647.238,Z 844.416,A 0.000,B 0.000,C 90.000,E1 290.844} C_DIS
LIN {X 0.032,Y -641.802,Z 844.415,A 0.000,B 0.000,C 90.000,E1 290.663} C_DIS
LIN {X 0.374,Y -638.146,Z 844.414,A 0.000,B 0.000,C 90.000,E1 290.482} C_DIS
LIN {X 0.168,Y -636.590,Z 844.414,A 0.000,B 0.000,C 90.000,E1 290.429} C_DIS
LIN {X 0.200,Y -633.867,Z 844.413,A 0.000,B 0.000,C 90.000,E1 290.248} C_DIS
LIN {X 0.166,Y -633.831,Z 844.413,A 0.000,B 0.000,C 90.000,E1 290.248} C_DIS
LIN {X 0.096,Y -632.793,Z 844.412,A 0.000,B 0.000,C 90.000,E1 290.066} C_DIS
LIN {X 0.053,Y -632.770,Z 844.412,A 0.000,B 0.000,C 90.000,E1 290.066} C_DIS
LIN {X -0.154,Y -632.948,Z 844.411,A 0.000,B 0.000,C 90.000,E1 289.939} C_DIS
LIN {X -0.145,Y -633.256,Z 844.410,A 0.000,B 0.000,C 90.000,E1 289.812} C_DIS
LIN {X 0.277,Y -635.255,Z 844.408,A 0.000,B 0.000,C 90.000,E1 289.322} C_DIS
LIN {X 0.047,Y -640.697,Z 844.402,A 0.000,B 0.000,C 90.000,E1 288.362} C_DIS
LIN {X -0.211,Y -643.894,Z 844.399,A 0.000,B 0.000,C 90.000,E1 287.764} C_DIS
LIN {X 0.138,Y -647.249,Z 844.394,A 0.000,B 0.000,C 90.000,E1 286.985} C_DIS
LIN {X -0.101,Y -650.137,Z 844.390,A 0.000,B 0.000,C 90.000,E1 286.260} C_DIS
LIN {X -0.368,Y -651.886,Z 844.388,A 0.000,B 0.000,C 90.000,E1 285.788} C_DIS
LIN {X 0.181,Y -653.452,Z 844.385,A 0.000,B 0.000,C 90.000,E1 285.245} C_DIS
LIN {X -0.181,Y -655.247,Z 844.381,A 0.000,B 0.000,C 90.000,E1 284.537} C_DIS
LIN {X 0.112,Y -656.637,Z 844.377,A 0.000,B 0.000,C 90.000,E1 283.772} C_DIS
LIN {X -0.107,Y -657.332,Z 844.374,A 0.000,B 0.000,C 90.000,E1 283.300} C_DIS
LIN {X -0.324,Y -657.786,Z 844.371,A 0.000,B 0.000,C 90.000,E1 282.827} C_DIS
LIN {X 0.103,Y -658.016,Z 844.368,A 0.000,B 0.000,C 90.000,E1 282.299} C_DIS
LIN {X -0.221,Y -657.948,Z 844.364,A 0.000,B 0.000,C 90.000,E1 281.591} C_DIS
LIN {X 0.077,Y -657.687,Z 844.362,A 0.000,B 0.000,C 90.000,E1 281.074} C_DIS
LIN {X -0.257,Y -656.841,Z 844.358,A 0.000,B 0.000,C 90.000,E1 280.366} C_DIS
LIN {X 0.045,Y -655.919,Z 844.355,A 0.000,B 0.000,C 90.000,E1 279.849} C_DIS
LIN {X -0.195,Y -654.776,Z 844.352,A 0.000,B 0.000,C 90.000,E1 279.378} C_DIS
LIN {X 0.098,Y -653.294,Z 844.349,A 0.000,B 0.000,C 90.000,E1 278.859} C_DIS
LIN {X -0.261,Y -651.342,Z 844.347,A 0.000,B 0.000,C 90.000,E1 278.398} C_DIS
LIN {X -0.012,Y -648.440,Z 844.343,A 0.000,B 0.000,C 90.000,E1 277.757} C_DIS
LIN {X 0.121,Y -644.829,Z 844.340,A 0.000,B 0.000,C 90.000,E1 277.125} C_DIS
LIN {X -0.288,Y -641.710,Z 844.337,A 0.000,B 0.000,C 90.000,E1 276.663} C_DIS
LIN {X -0.080,Y -637.726,Z 844.334,A 0.000,B 0.000,C 90.000,E1 276.144} C_DIS
LIN {X 0.099,Y -633.332,Z 844.331,A 0.000,B 0.000,C 90.000,E1 275.625} C_DIS
LIN {X -0.033,Y -632.003,Z 844.331,A 0.000,B 0.000,C 90.000,E1 275.511} C_DIS
LIN {X -0.022,Y -627.956,Z 844.329,A 0.000,B 0.000,C 90.000,E1 275.163} C_DIS
LIN {X 0.246,Y -625.679,Z 844.328,A 0.000,B 0.000,C 90.000,E1 274.935} C_DIS
LIN {X -0.288,Y -618.183,Z 844.325,A 0.000,B 0.000,C 90.000,E1 274.473} C_DIS
LIN {X 0.109,Y -611.902,Z 844.323,A 0.000,B 0.000,C 90.000,E1 274.073} C_DIS
LIN {X 0.186,Y -605.144,Z 844.321,A 0.000,B 0.000,C 90.000,E1 273.726} C_DIS
LIN {X -0.125,Y -598.527,Z 844.319,A 0.000,B 0.000,C 90.000,E1 273.440} C_DIS
LIN {X -0.062,Y -589.618,Z 844.317,A 0.000,B 0.000,C 90.000,E1 273.094} C_DIS
LIN {X -0.228,Y -584.185,Z 844.316,A 0.000,B 0.000,C 90.000,E1 272.922} C_DIS
LIN {X -0.012,Y -578.022,Z 844.315,A 0.000,B 0.000,C 90.000,E1 272.751} C_DIS
LIN {X 0.280,Y -572.903,Z 844.315,A 0.000,B 0.000,C 90.000,E1 272.636} C_DIS
LIN {X 0.258,Y -567.057,Z 844.315,A 0.000,B 0.000,C 90.000,E1 272.579} C_DIS
LIN {X 0.024,Y -563.084,Z 844.314,A 0.000,B 0.000,C 90.000,E1 272.579} C_DIS
LIN {X -0.115,Y -557.218,Z 844.314,A 0.000,B 0.000,C 90.000,E1 272.579} C_DIS
LIN {X 0.183,Y -553.688,Z 844.314,A 0.000,B 0.000,C 90.000,E1 272.522} C_DIS
LIN {X 0.178,Y -550.458,Z 844.314,A 0.000,B 0.000,C 90.000,E1 272.407} C_DIS
LIN {X 0.139,Y -550.398,Z 844.313,A 0.000,B 0.000,C 90.000,E1 272.407} C_DIS
LIN {X 0.127,Y -549.119,Z 844.312,A 0.000,B 0.000,C 90.000,E1 272.178} C_DIS
LIN {X 0.181,Y -548.282,Z 844.311,A 0.000,B 0.000,C 90.000,E1 271.892} C_DIS
LIN {X -0.003,Y -547.481,Z 844.308,A 0.000,B 0.000,C 90.000,E1 271.489} C_DIS
LIN {X 0.180,Y -546.216,Z 844.302,A 0.000,B 0.000,C 90.000,E1 270.344} C_DIS
LIN {X -0.086,Y -544.700,Z 844.291,A 0.000,B 0.000,C 90.000,E1 268.396} C_DIS
LIN {X 0.099,Y -543.714,Z 844.283,A 0.000,B 0.000,C 90.000,E1 266.963} C_DIS
LIN {X -0.220,Y -542.537,Z 844.274,A 0.000,B 0.000,C 90.000,E1 265.298} C_DIS
LIN {X 0.013,Y -541.584,Z 844.266,A 0.000,B 0.000,C 90.000,E1 263.856} C_DIS
LIN {X 0.096,Y -540.881,Z 844.261,A 0.000,B 0.000,C 90.000,E1 262.996} C_DIS
LIN {X -0.092,Y -539.342,Z 844.252,A 0.000,B 0.000,C 90.000,E1 261.310} C_DIS
LIN {X 0.165,Y -538.012,Z 844.244,A 0.000,B 0.000,C 90.000,E1 259.859} C_DIS
LIN {X -0.080,Y -536.270,Z 844.234,A 0.000,B 0.000,C 90.000,E1 258.173} C_DIS
LIN {X -0.198,Y -534.791,Z 844.226,A 0.000,B 0.000,C 90.000,E1 256.756} C_DIS
LIN {X 0.182,Y -533.123,Z 844.218,A 0.000,B 0.000,C 90.000,E1 255.283} C_DIS
LIN {X 0.005,Y -531.467,Z 844.210,A 0.000,B 0.000,C 90.000,E1 253.866} C_DIS
LIN {X 0.094,Y -529.773,Z 844.202,A 0.000,B 0.000,C 90.000,E1 252.417} C_DIS
LIN {X 0.162,Y -527.947,Z 844.194,A 0.000,B 0.000,C 90.000,E1 250.967} C_DIS
LIN {X 0.015,Y -526.436,Z 844.188,A 0.000,B 0.000,C 90.000,E1 249.826} C_DIS
LIN {X -0.301,Y -524.452,Z 844.180,A 0.000,B 0.000,C 90.000,E1 248.411} C_DIS
LIN {X 0.188,Y -521.961,Z 844.170,A 0.000,B 0.000,C 90.000,E1 246.613} C_DIS
LIN {X -0.155,Y -520.221,Z 844.164,A 0.000,B 0.000,C 90.000,E1 245.485} C_DIS
LIN {X -0.165,Y -517.873,Z 844.156,A 0.000,B 0.000,C 90.000,E1 244.024} C_DIS
LIN {X 0.130,Y -514.797,Z 844.146,A 0.000,B 0.000,C 90.000,E1 242.231} C_DIS
LIN {X -0.214,Y -511.148,Z 844.134,A 0.000,B 0.000,C 90.000,E1 240.205} C_DIS
LIN {X -0.135,Y -507.270,Z 844.123,A 0.000,B 0.000,C 90.000,E1 238.122} C_DIS
LIN {X 0.023,Y -504.904,Z 844.116,A 0.000,B 0.000,C 90.000,E1 236.914} C_DIS
LIN {X 0.001,Y -502.337,Z 844.110,A 0.000,B 0.000,C 90.000,E1 235.722} C_DIS
LIN {X -0.053,Y -499.644,Z 844.103,A 0.000,B 0.000,C 90.000,E1 234.529} C_DIS
LIN {X 0.006,Y -493.911,Z 844.090,A 0.000,B 0.000,C 90.000,E1 232.110} C_DIS
LIN {X 0.113,Y -491.121,Z 844.083,A 0.000,B 0.000,C 90.000,E1 230.884} C_DIS
LIN {X 0.094,Y -486.889,Z 844.073,A 0.000,B 0.000,C 90.000,E1 229.057} C_DIS
LIN {X 0.033,Y -484.036,Z 844.066,A 0.000,B 0.000,C 90.000,E1 227.838} C_DIS
LIN {X -0.031,Y -479.339,Z 844.054,A 0.000,B 0.000,C 90.000,E1 225.688} C_DIS
LIN {X 0.217,Y -475.995,Z 844.045,A 0.000,B 0.000,C 90.000,E1 224.109} C_DIS
LIN {X -0.082,Y -471.241,Z 844.033,A 0.000,B 0.000,C 90.000,E1 221.962} C_DIS
LIN {X -0.027,Y -468.540,Z 844.026,A 0.000,B 0.000,C 90.000,E1 220.701} C_DIS
LIN {X -0.188,Y -464.654,Z 844.016,A 0.000,B 0.000,C 90.000,E1 218.830} C_DIS
LIN {X 0.136,Y -461.987,Z 844.009,A 0.000,B 0.000,C 90.000,E1 217.523} C_DIS
LIN {X 0.153,Y -458.751,Z 844.000,A 0.000,B 0.000,C 90.000,E1 215.931} C_DIS
LIN {X 0.029,Y -453.889,Z 843.987,A 0.000,B 0.000,C 90.000,E1 213.706} C_DIS
LIN {X -0.093,Y -449.096,Z 843.975,A 0.000,B 0.000,C 90.000,E1 211.465} C_DIS
LIN {X -0.195,Y -444.331,Z 843.962,A 0.000,B 0.000,C 90.000,E1 209.205} C_DIS
LIN {X -0.184,Y -441.709,Z 843.955,A 0.000,B 0.000,C 90.000,E1 207.897} C_DIS
LIN {X 0.036,Y -437.777,Z 843.944,A 0.000,B 0.000,C 90.000,E1 205.899} C_DIS
LIN {X -0.053,Y -435.050,Z 843.937,A 0.000,B 0.000,C 90.000,E1 204.591} C_DIS
LIN {X -0.180,Y -431.664,Z 843.927,A 0.000,B 0.000,C 90.000,E1 202.950} C_DIS
LIN {X 0.055,Y -427.786,Z 843.916,A 0.000,B 0.000,C 90.000,E1 200.918} C_DIS
LIN {X -0.164,Y -423.227,Z 843.903,A 0.000,B 0.000,C 90.000,E1 198.598} C_DIS
LIN {X 0.026,Y -418.632,Z 843.890,A 0.000,B 0.000,C 90.000,E1 196.205} C_DIS
LIN {X -0.006,Y -416.676,Z 843.884,A 0.000,B 0.000,C 90.000,E1 195.190} C_DIS
LIN {X -0.025,Y -413.906,Z 843.877,A 0.000,B 0.000,C 90.000,E1 193.828} C_DIS
LIN {X -0.008,Y -409.154,Z 843.864,A 0.000,B 0.000,C 90.000,E1 191.422} C_DIS
LIN {X 0.169,Y -405.868,Z 843.854,A 0.000,B 0.000,C 90.000,E1 189.670} C_DIS
LIN {X 0.145,Y -402.524,Z 843.844,A 0.000,B 0.000,C 90.000,E1 187.936} C_DIS
LIN {X -0.046,Y -397.204,Z 843.829,A 0.000,B 0.000,C 90.000,E1 185.163} C_DIS
LIN {X -0.116,Y -392.675,Z 843.813,A 0.000,B 0.000,C 90.000,E1 182.350} C_DIS
LIN {X -0.147,Y -387.794,Z 843.793,A 0.000,B 0.000,C 90.000,E1 178.797} C_DIS
LIN {X 0.150,Y -385.321,Z 843.783,A 0.000,B 0.000,C 90.000,E1 176.963} C_DIS
LIN {X -0.059,Y -382.574,Z 843.771,A 0.000,B 0.000,C 90.000,E1 174.837} C_DIS
LIN {X 0.084,Y -379.883,Z 843.759,A 0.000,B 0.000,C 90.000,E1 172.648} C_DIS
LIN {X -0.047,Y -376.331,Z 843.741,A 0.000,B 0.000,C 90.000,E1 169.398} C_DIS
LIN {X -0.093,Y -373.545,Z 843.723,A 0.000,B 0.000,C 90.000,E1 166.117} C_DIS
LIN {X -0.155,Y -372.097,Z 843.709,A 0.000,B 0.000,C 90.000,E1 163.559} C_DIS
LIN {X 0.102,Y -371.875,Z 843.702,A 0.000,B 0.000,C 90.000,E1 162.417} C_DIS
LIN {X 0.004,Y -372.038,Z 843.696,A 0.000,B 0.000,C 90.000,E1 161.329} C_DIS
LIN {X -0.061,Y -372.288,Z 843.692,A 0.000,B 0.000,C 90.000,E1 160.604} C_DIS
LIN {X -0.127,Y -372.723,Z 843.688,A 0.000,B 0.000,C 90.000,E1 159.880} C_DIS
LIN {X -0.055,Y -374.027,Z 843.682,A 0.000,B 0.000,C 90.000,E1 158.773} C_DIS
LIN {X 0.025,Y -375.166,Z 843.678,A 0.000,B 0.000,C 90.000,E1 158.028} C_DIS
LIN {X 0.105,Y -377.145,Z 843.673,A 0.000,B 0.000,C 90.000,E1 157.102} C_DIS
LIN {X 0.071,Y -378.814,Z 843.670,A 0.000,B 0.000,C 90.000,E1 156.561} C_DIS
LIN {X 0.091,Y -381.455,Z 843.667,A 0.000,B 0.000,C 90.000,E1 155.973} C_DIS
LIN {X -0.112,Y -386.011,Z 843.663,A 0.000,B 0.000,C 90.000,E1 155.281} C_DIS
LIN {X 0.159,Y -387.072,Z 843.662,A 0.000,B 0.000,C 90.000,E1 155.101} C_DIS
LIN {X 0.081,Y -388.442,Z 843.661,A 0.000,B 0.000,C 90.000,E1 154.973} C_DIS
LIN {X -0.164,Y -393.822,Z 843.659,A 0.000,B 0.000,C 90.000,E1 154.588} C_DIS
LIN {X 0.103,Y -397.798,Z 843.658,A 0.000,B 0.000,C 90.000,E1 154.332} C_DIS
LIN {X 0.148,Y -401.556,Z 843.657,A 0.000,B 0.000,C 90.000,E1 154.152} C_DIS
LIN {X 0.048,Y -412.421,Z 843.654,A 0.000,B 0.000,C 90.000,E1 153.768} C_DIS
LIN {X 0.010,Y -415.829,Z 843.654,A 0.000,B 0.000,C 90.000,E1 153.640} C_DIS
LIN {X 0.227,Y -425.754,Z 843.651,A 0.000,B 0.000,C 90.000,E1 153.127} C_DIS
LIN {X 0.014,Y -435.655,Z 843.648,A 0.000,B 0.000,C 90.000,E1 152.615} C_DIS
LIN {X 0.040,Y -438.538,Z 843.647,A 0.000,B 0.000,C 90.000,E1 152.436} C_DIS
LIN {X 0.158,Y -443.007,Z 843.645,A 0.000,B 0.000,C 90.000,E1 152.103} C_DIS
LIN {X -0.130,Y -444.768,Z 843.645,A 0.000,B 0.000,C 90.000,E1 152.025} C_DIS
LIN {X 0.041,Y -452.322,Z 843.641,A 0.000,B 0.000,C 90.000,E1 151.435} C_DIS
LIN {X -0.074,Y -456.868,Z 843.639,A 0.000,B 0.000,C 90.000,E1 151.101} C_DIS
LIN {X -0.241,Y -465.305,Z 843.635,A 0.000,B 0.000,C 90.000,E1 150.333} C_DIS
LIN {X -0.071,Y -473.588,Z 843.630,A 0.000,B 0.000,C 90.000,E1 149.459} C_DIS
LIN {X 0.120,Y -480.215,Z 843.626,A 0.000,B 0.000,C 90.000,E1 148.742} C_DIS
LIN {X -0.303,Y -485.546,Z 843.623,A 0.000,B 0.000,C 90.000,E1 148.201} C_DIS
LIN {X -0.181,Y -490.569,Z 843.620,A 0.000,B 0.000,C 90.000,E1 147.582} C_DIS
LIN {X 0.176,Y -497.584,Z 843.615,A 0.000,B 0.000,C 90.000,E1 146.628} C_DIS
LIN {X -0.171,Y -500.901,Z 843.612,A 0.000,B 0.000,C 90.000,E1 146.215} C_DIS
LIN {X -0.082,Y -504.175,Z 843.610,A 0.000,B 0.000,C 90.000,E1 145.754} C_DIS
LIN {X -0.088,Y -511.620,Z 843.603,A 0.000,B 0.000,C 90.000,E1 144.562} C_DIS
LIN {X 0.017,Y -518.683,Z 843.597,A 0.000,B 0.000,C 90.000,E1 143.371} C_DIS
LIN {X -0.091,Y -528.220,Z 843.588,A 0.000,B 0.000,C 90.000,E1 141.778} C_DIS
LIN {X -0.259,Y -537.933,Z 843.578,A 0.000,B 0.000,C 90.000,E1 140.070} C_DIS
LIN {X -0.058,Y -546.348,Z 843.569,A 0.000,B 0.000,C 90.000,E1 138.485} C_DIS
LIN {X 0.210,Y -551.541,Z 843.564,A 0.000,B 0.000,C 90.000,E1 137.472} C_DIS
LIN {X -0.237,Y -556.642,Z 843.558,A 0.000,B 0.000,C 90.000,E1 136.539} C_DIS
LIN {X -0.134,Y -559.736,Z 843.555,A 0.000,B 0.000,C 90.000,E1 135.972} C_DIS
LIN {X 0.067,Y -563.872,Z 843.551,A 0.000,B 0.000,C 90.000,E1 135.121} C_DIS
LIN {X 0.004,Y -569.205,Z 843.545,A 0.000,B 0.000,C 90.000,E1 134.028} C_DIS
LIN {X 0.254,Y -576.944,Z 843.536,A 0.000,B 0.000,C 90.000,E1 132.366} C_DIS
LIN {X 0.106,Y -581.197,Z 843.530,A 0.000,B 0.000,C 90.000,E1 131.434} C_DIS
LIN {X 0.076,Y -587.045,Z 843.523,A 0.000,B 0.000,C 90.000,E1 130.092} C_DIS
LIN {X 0.147,Y -592.537,Z 843.515,A 0.000,B 0.000,C 90.000,E1 128.749} C_DIS
LIN {X -0.289,Y -596.213,Z 843.510,A 0.000,B 0.000,C 90.000,E1 127.729} C_DIS
LIN {X -0.078,Y -598.737,Z 843.505,A 0.000,B 0.000,C 90.000,E1 126.916} C_DIS
LIN {X 0.283,Y -601.045,Z 843.501,A 0.000,B 0.000,C 90.000,E1 126.091} C_DIS
LIN {X -0.400,Y -603.661,Z 843.495,A 0.000,B 0.000,C 90.000,E1 125.105} C_DIS
LIN {X 0.025,Y -605.327,Z 843.490,A 0.000,B 0.000,C 90.000,E1 124.278} C_DIS
LIN {X -0.103,Y -607.160,Z 843.485,A 0.000,B 0.000,C 90.000,E1 123.245} C_DIS
LIN {X 0.057,Y -609.186,Z 843.477,A 0.000,B 0.000,C 90.000,E1 121.926} C_DIS
LIN {X 0.170,Y -610.442,Z 843.472,A 0.000,B 0.000,C 90.000,E1 120.875} C_DIS
LIN {X -0.220,Y -611.516,Z 843.466,A 0.000,B 0.000,C 90.000,E1 119.873} C_DIS
LIN {X -0.068,Y -612.091,Z 843.460,A 0.000,B 0.000,C 90.000,E1 118.821} C_DIS
LIN {X 0.156,Y -612.284,Z 843.457,A 0.000,B 0.000,C 90.000,E1 118.281} C_DIS
LIN {X 0.056,Y -612.262,Z 843.453,A 0.000,B 0.000,C 90.000,E1 117.513} C_DIS
LIN {X -0.007,Y -612.095,Z 843.450,A 0.000,B 0.000,C 90.000,E1 117.001} C_DIS
LIN {X -0.173,Y -611.089,Z 843.443,A 0.000,B 0.000,C 90.000,E1 115.720} C_DIS
LIN {X -0.245,Y -610.529,Z 843.440,A 0.000,B 0.000,C 90.000,E1 115.207} C_DIS
LIN {X 0.231,Y -609.671,Z 843.437,A 0.000,B 0.000,C 90.000,E1 114.643} C_DIS
LIN {X 0.146,Y -608.637,Z 843.434,A 0.000,B 0.000,C 90.000,E1 114.131} C_DIS
LIN {X -0.243,Y -606.488,Z 843.430,A 0.000,B 0.000,C 90.000,E1 113.387} C_DIS
LIN {X 0.204,Y -604.762,Z 843.427,A 0.000,B 0.000,C 90.000,E1 112.823} C_DIS
LIN {X -0.089,Y -603.204,Z 843.425,A 0.000,B 0.000,C 90.000,E1 112.589} C_DIS
LIN {X -0.154,Y -601.991,Z 843.424,A 0.000,B 0.000,C 90.000,E1 112.333} C_DIS
LIN {X -0.224,Y -599.590,Z 843.423,A 0.000,B 0.000,C 90.000,E1 112.078} C_DIS
LIN {X -0.274,Y -598.314,Z 843.422,A 0.000,B 0.000,C 90.000,E1 111.897} C_DIS
LIN {X 0.239,Y -597.161,Z 843.421,A 0.000,B 0.000,C 90.000,E1 111.716} C_DIS
LIN {X -0.199,Y -591.366,Z 843.418,A 0.000,B 0.000,C 90.000,E1 111.280} C_DIS
LIN {X 0.064,Y -584.913,Z 843.416,A 0.000,B 0.000,C 90.000,E1 110.844} C_DIS
LIN {X 0.071,Y -574.379,Z 843.413,A 0.000,B 0.000,C 90.000,E1 110.355} C_DIS
LIN {X 0.161,Y -570.854,Z 843.412,A 0.000,B 0.000,C 90.000,E1 110.194} C_DIS
LIN {X 0.168,Y -569.659,Z 843.412,A 0.000,B 0.000,C 90.000,E1 110.120} C_DIS
LIN {X 0.152,Y -565.652,Z 843.410,A 0.000,B 0.000,C 90.000,E1 109.758} C_DIS
LIN {X 0.115,Y -565.623,Z 843.410,A 0.000,B 0.000,C 90.000,E1 109.758} C_DIS
LIN {X 0.011,Y -564.393,Z 843.408,A 0.000,B 0.000,C 90.000,E1 109.504} C_DIS
LIN {X -0.279,Y -563.754,Z 843.408,A 0.000,B 0.000,C 90.000,E1 109.396} C_DIS
LIN {X -0.133,Y -562.985,Z 843.406,A 0.000,B 0.000,C 90.000,E1 109.033} C_DIS
LIN {X -0.240,Y -562.512,Z 843.405,A 0.000,B 0.000,C 90.000,E1 108.906} C_DIS
LIN {X 0.125,Y -561.746,Z 843.402,A 0.000,B 0.000,C 90.000,E1 108.308} C_DIS
LIN {X -0.051,Y -561.166,Z 843.396,A 0.000,B 0.000,C 90.000,E1 107.221} C_DIS
LIN {X -0.304,Y -561.474,Z 843.380,A 0.000,B 0.000,C 90.000,E1 104.481} C_DIS
LIN {X -0.032,Y -562.548,Z 843.368,A 0.000,B 0.000,C 90.000,E1 102.243} C_DIS
LIN {X -0.017,Y -563.849,Z 843.357,A 0.000,B 0.000,C 90.000,E1 100.310} C_DIS
LIN {X 0.308,Y -565.021,Z 843.348,A 0.000,B 0.000,C 90.000,E1 98.624} C_DIS
LIN {X -0.153,Y -565.936,Z 843.341,A 0.000,B 0.000,C 90.000,E1 97.296} C_DIS
LIN {X 0.065,Y -566.875,Z 843.331,A 0.000,B 0.000,C 90.000,E1 95.625} C_DIS
LIN {X -0.124,Y -567.269,Z 843.327,A 0.000,B 0.000,C 90.000,E1 94.821} C_DIS
LIN {X 0.080,Y -567.928,Z 843.318,A 0.000,B 0.000,C 90.000,E1 93.154} C_DIS
LIN {X 0.163,Y -568.324,Z 843.310,A 0.000,B 0.000,C 90.000,E1 91.776} C_DIS
LIN {X -0.232,Y -568.777,Z 843.301,A 0.000,B 0.000,C 90.000,E1 90.172} C_DIS
LIN {X 0.077,Y -569.288,Z 843.290,A 0.000,B 0.000,C 90.000,E1 88.224} C_DIS
LIN {X -0.260,Y -569.552,Z 843.281,A 0.000,B 0.000,C 90.000,E1 86.617} C_DIS
LIN {X -0.013,Y -569.839,Z 843.272,A 0.000,B 0.000,C 90.000,E1 84.951} C_DIS
LIN {X 0.111,Y -570.117,Z 843.264,A 0.000,B 0.000,C 90.000,E1 83.571} C_DIS
LIN {X 0.203,Y -570.658,Z 843.252,A 0.000,B 0.000,C 90.000,E1 81.376} C_DIS
LIN {X 0.125,Y -571.417,Z 843.239,A 0.000,B 0.000,C 90.000,E1 78.926} C_DIS
LIN {X -0.147,Y -571.880,Z 843.231,A 0.000,B 0.000,C 90.000,E1 77.589} C_DIS
LIN {X 0.024,Y -572.354,Z 843.222,A 0.000,B 0.000,C 90.000,E1 75.936} C_DIS
LIN {X 0.018,Y -572.633,Z 843.214,A 0.000,B 0.000,C 90.000,E1 74.574} C_DIS
LIN {X 0.172,Y -572.797,Z 843.207,A 0.000,B 0.000,C 90.000,E1 73.196} C_DIS
LIN {X -0.204,Y -572.807,Z 843.202,A 0.000,B 0.000,C 90.000,E1 72.417} C_DIS
LIN {X -0.235,Y -572.843,Z 843.193,A 0.000,B 0.000,C 90.000,E1 70.786} C_DIS
LIN {X -0.076,Y -572.679,Z 843.184,A 0.000,B 0.000,C 90.000,E1 69.135} C_DIS
LIN {X -0.097,Y -572.413,Z 843.174,A 0.000,B 0.000,C 90.000,E1 67.230} C_DIS
LIN {X -0.110,Y -572.131,Z 843.166,A 0.000,B 0.000,C 90.000,E1 65.869} C_DIS
LIN {X 0.096,Y -571.624,Z 843.158,A 0.000,B 0.000,C 90.000,E1 64.485} C_DIS
LIN {X 0.029,Y -571.113,Z 843.151,A 0.000,B 0.000,C 90.000,E1 63.127} C_DIS
LIN {X -0.038,Y -570.587,Z 843.143,A 0.000,B 0.000,C 90.000,E1 61.769} C_DIS
LIN {X 0.225,Y -570.168,Z 843.139,A 0.000,B 0.000,C 90.000,E1 60.923} C_DIS
LIN {X -0.188,Y -569.378,Z 843.133,A 0.000,B 0.000,C 90.000,E1 59.871} C_DIS
LIN {X 0.162,Y -568.359,Z 843.126,A 0.000,B 0.000,C 90.000,E1 58.742} C_DIS
LIN {X 0.011,Y -567.139,Z 843.120,A 0.000,B 0.000,C 90.000,E1 57.661} C_DIS
LIN {X -0.158,Y -565.791,Z 843.114,A 0.000,B 0.000,C 90.000,E1 56.580} C_DIS
LIN {X -0.036,Y -564.157,Z 843.108,A 0.000,B 0.000,C 90.000,E1 55.468} C_DIS
LIN {X -0.041,Y -562.819,Z 843.104,A 0.000,B 0.000,C 90.000,E1 54.642} C_DIS
LIN {X -0.190,Y -561.293,Z 843.099,A 0.000,B 0.000,C 90.000,E1 53.829} C_DIS
LIN {X -0.138,Y -558.930,Z 843.093,A 0.000,B 0.000,C 90.000,E1 52.718} C_DIS
LIN {X -0.315,Y -556.974,Z 843.088,A 0.000,B 0.000,C 90.000,E1 51.904} C_DIS
LIN {X -0.151,Y -555.555,Z 843.085,A 0.000,B 0.000,C 90.000,E1 51.331} C_DIS
LIN {X -0.007,Y -553.128,Z 843.081,A 0.000,B 0.000,C 90.000,E1 50.481} C_DIS
LIN {X 0.183,Y -550.394,Z 843.076,A 0.000,B 0.000,C 90.000,E1 49.622} C_DIS
LIN {X -0.128,Y -548.391,Z 843.073,A 0.000,B 0.000,C 90.000,E1 49.094} C_DIS
LIN {X -0.054,Y -545.031,Z 843.068,A 0.000,B 0.000,C 90.000,E1 48.243} C_DIS
LIN {X -0.206,Y -541.989,Z 843.064,A 0.000,B 0.000,C 90.000,E1 47.553} C_DIS
LIN {X -0.209,Y -539.341,Z 843.061,A 0.000,B 0.000,C 90.000,E1 46.986} C_DIS
LIN {X 0.161,Y -536.516,Z 843.058,A 0.000,B 0.000,C 90.000,E1 46.377} C_DIS
LIN {X 0.118,Y -533.388,Z 843.055,A 0.000,B 0.000,C 90.000,E1 45.810} C_DIS
LIN {X 0.223,Y -528.956,Z 843.051,A 0.000,B 0.000,C 90.000,E1 45.081} C_DIS
LIN {X 0.129,Y -525.093,Z 843.047,A 0.000,B 0.000,C 90.000,E1 44.514} C_DIS
LIN {X 0.069,Y -521.013,Z 843.044,A 0.000,B 0.000,C 90.000,E1 43.947} C_DIS
LIN {X -0.083,Y -516.499,Z 843.041,A 0.000,B 0.000,C 90.000,E1 43.380} C_DIS
LIN {X -0.025,Y -513.011,Z 843.039,A 0.000,B 0.000,C 90.000,E1 42.933} C_DIS
LIN {X -0.048,Y -508.127,Z 843.035,A 0.000,B 0.000,C 90.000,E1 42.366} C_DIS
LIN {X 0.324,Y -502.942,Z 843.032,A 0.000,B 0.000,C 90.000,E1 41.757} C_DIS
LIN {X -0.148,Y -498.976,Z 843.030,A 0.000,B 0.000,C 90.000,E1 41.391} C_DIS
LIN {X -0.142,Y -491.986,Z 843.026,A 0.000,B 0.000,C 90.000,E1 40.701} C_DIS
LIN {X 0.178,Y -487.457,Z 843.024,A 0.000,B 0.000,C 90.000,E1 40.253} C_DIS
LIN {X 0.020,Y -480.205,Z 843.020,A 0.000,B 0.000,C 90.000,E1 39.644} C_DIS
LIN {X -0.125,Y -472.531,Z 843.017,A 0.000,B 0.000,C 90.000,E1 39.036} C_DIS
LIN {X 0.044,Y -463.371,Z 843.013,A 0.000,B 0.000,C 90.000,E1 38.302} C_DIS
LIN {X 0.180,Y -452.398,Z 843.008,A 0.000,B 0.000,C 90.000,E1 37.443} C_DIS
LIN {X -0.167,Y -434.997,Z 843.001,A 0.000,B 0.000,C 90.000,E1 36.171} C_DIS
LIN {X -0.204,Y -413.457,Z 842.991,A 0.000,B 0.000,C 90.000,E1 34.405} C_DIS
LIN {X -0.249,Y -404.514,Z 842.986,A 0.000,B 0.000,C 90.000,E1 33.579} C_DIS
LIN {X 0.063,Y -400.158,Z 842.984,A 0.000,B 0.000,C 90.000,E1 33.086} C_DIS
LIN {X 0.208,Y -397.477,Z 842.982,A 0.000,B 0.000,C 90.000,E1 32.752} C_DIS
LIN {X -0.196,Y -394.480,Z 842.980,A 0.000,B 0.000,C 90.000,E1 32.339} C_DIS
LIN {X 0.100,Y -394.450,Z 842.980,A 0.000,B 0.000,C 90.000,E1 32.291} C_DIS
LIN {X 0.110,Y -393.517,Z 842.976,A 0.000,B 0.000,C 90.000,E1 31.671} C_DIS
LIN {X 0.089,Y -390.798,Z 842.968,A 0.000,B 0.000,C 90.000,E1 30.256} C_DIS
LIN {X -0.058,Y -390.732,Z 842.966,A 0.000,B 0.000,C 90.000,E1 29.922} C_DIS
LIN {X 0.068,Y -393.185,Z 842.941,A 0.000,B 0.000,C 90.000,E1 25.283} C_DIS
LIN {X -0.055,Y -395.077,Z 842.927,A 0.000,B 0.000,C 90.000,E1 22.823} C_DIS
LIN {X -0.076,Y -397.229,Z 842.913,A 0.000,B 0.000,C 90.000,E1 20.355} C_DIS
LIN {X 0.105,Y -400.516,Z 842.896,A 0.000,B 0.000,C 90.000,E1 17.166} C_DIS
LIN {X 0.206,Y -404.056,Z 842.880,A 0.000,B 0.000,C 90.000,E1 14.356} C_DIS
LIN {X 0.109,Y -408.163,Z 842.865,A 0.000,B 0.000,C 90.000,E1 11.591} C_DIS
LIN {X -0.159,Y -411.531,Z 842.853,A 0.000,B 0.000,C 90.000,E1 9.557} C_DIS
LIN {X 0.019,Y -414.481,Z 842.844,A 0.000,B 0.000,C 90.000,E1 7.814} C_DIS
LIN {X 0.200,Y -418.142,Z 842.832,A 0.000,B 0.000,C 90.000,E1 5.739} C_DIS
LIN {X 0.049,Y -422.582,Z 842.819,A 0.000,B 0.000,C 90.000,E1 3.383} C_DIS
LIN {X 0.000,Y -429.775,Z 842.800,A 0.000,B 0.000,C 90.000,E1 360.000} C_DIS
LIN {X -0.119,Y -435.771,Z 842.786,A 0.000,B 0.000,C 90.000,E1 357.478} C_DIS
LIN {X -0.013,Y -439.814,Z 842.777,A 0.000,B 0.000,C 90.000,E1 355.812} C_DIS
LIN {X -0.089,Y -447.620,Z 842.760,A 0.000,B 0.000,C 90.000,E1 352.875} C_DIS
LIN {X 0.094,Y -449.955,Z 842.757,A 0.000,B 0.000,C 90.000,E1 352.243} C_DIS
LIN {X -0.096,Y -452.517,Z 842.754,A 0.000,B 0.000,C 90.000,E1 351.781} C_DIS
LIN {X 0.037,Y -453.677,Z 842.753,A 0.000,B 0.000,C 90.000,E1 351.602} C_DIS
LIN {X 0.107,Y -456.700,Z 842.752,A 0.000,B 0.000,C 90.000,E1 351.319} C_DIS
LIN {X -0.059,Y -458.700,Z 842.751,A 0.000,B 0.000,C 90.000,E1 351.141} C_DIS
LIN {X -0.138,Y -459.522,Z 842.750,A 0.000,B 0.000,C 90.000,E1 351.084} C_DIS
LIN {X 0.084,Y -467.828,Z 842.748,A 0.000,B 0.000,C 90.000,E1 350.557} C_DIS
LIN {X 0.078,Y -472.994,Z 842.746,A 0.000,B 0.000,C 90.000,E1 350.274} C_DIS
LIN {X -0.156,Y -477.986,Z 842.745,A 0.000,B 0.000,C 90.000,E1 350.038} C_DIS
LIN {X 0.014,Y -487.633,Z 842.741,A 0.000,B 0.000,C 90.000,E1 349.454} C_DIS
LIN {X 0.052,Y -498.857,Z 842.738,A 0.000,B 0.000,C 90.000,E1 348.757} C_DIS
LIN {X -0.238,Y -506.649,Z 842.735,A 0.000,B 0.000,C 90.000,E1 348.285} C_DIS
LIN {X -0.041,Y -519.181,Z 842.730,A 0.000,B 0.000,C 90.000,E1 347.409} C_DIS
LIN {X -0.090,Y -528.242,Z 842.726,A 0.000,B 0.000,C 90.000,E1 346.756} C_DIS
LIN {X -0.002,Y -537.205,Z 842.723,A 0.000,B 0.000,C 90.000,E1 346.061} C_DIS
LIN {X 0.069,Y -545.850,Z 842.719,A 0.000,B 0.000,C 90.000,E1 345.353} C_DIS
LIN {X -0.037,Y -552.765,Z 842.715,A 0.000,B 0.000,C 90.000,E1 344.755} C_DIS
LIN {X -0.286,Y -559.392,Z 842.712,A 0.000,B 0.000,C 90.000,E1 344.157} C_DIS
LIN {X -0.078,Y -564.550,Z 842.709,A 0.000,B 0.000,C 90.000,E1 343.614} C_DIS
LIN {X -0.187,Y -569.538,Z 842.706,A 0.000,B 0.000,C 90.000,E1 343.087} C_DIS
LIN {X 0.225,Y -575.513,Z 842.702,A 0.000,B 0.000,C 90.000,E1 342.362} C_DIS
LIN {X -0.230,Y -578.920,Z 842.700,A 0.000,B 0.000,C 90.000,E1 342.000} C_DIS
LIN {X 0.275,Y -584.166,Z 842.696,A 0.000,B 0.000,C 90.000,E1 341.275} C_DIS
LIN {X 0.013,Y -590.188,Z 842.692,A 0.000,B 0.000,C 90.000,E1 340.496} C_DIS
LIN {X 0.061,Y -594.576,Z 842.688,A 0.000,B 0.000,C 90.000,E1 339.826} C_DIS
LIN {X 0.057,Y -600.365,Z 842.683,A 0.000,B 0.000,C 90.000,E1 338.901} C_DIS
LIN {X 0.157,Y -605.036,Z 842.678,A 0.000,B 0.000,C 90.000,E1 338.103} C_DIS
LIN {X 0.255,Y -610.976,Z 842.673,A 0.000,B 0.000,C 90.000,E1 337.050} C_DIS
LIN {X -0.102,Y -615.249,Z 842.668,A 0.000,B 0.000,C 90.000,E1 336.305} C_DIS
LIN {X -0.177,Y -619.945,Z 842.663,A 0.000,B 0.000,C 90.000,E1 335.409} C_DIS
LIN {X 0.110,Y -624.413,Z 842.658,A 0.000,B 0.000,C 90.000,E1 334.485} C_DIS
LIN {X 0.148,Y -628.652,Z 842.653,A 0.000,B 0.000,C 90.000,E1 333.589} C_DIS
LIN {X -0.348,Y -632.026,Z 842.649,A 0.000,B 0.000,C 90.000,E1 332.871} C_DIS
LIN {X -0.206,Y -636.296,Z 842.644,A 0.000,B 0.000,C 90.000,E1 331.847} C_DIS
LIN {X -0.208,Y -641.347,Z 842.637,A 0.000,B 0.000,C 90.000,E1 330.589} C_DIS
LIN {X 0.301,Y -644.265,Z 842.632,A 0.000,B 0.000,C 90.000,E1 329.793} C_DIS
LIN {X 0.028,Y -647.847,Z 842.627,A 0.000,B 0.000,C 90.000,E1 328.820} C_DIS
LIN {X 0.046,Y -650.409,Z 842.623,A 0.000,B 0.000,C 90.000,E1 328.074} C_DIS
